SPLINE
SPL {X  -160.133, Y  +702.956, Z    +0.000, E1   -19.806, E3 +417494.548}
SPL {X  -161.979, Y  +690.023, Z    +0.000, E1   -12.991, E3 +417497.464}
SPL {X  -162.641, Y  +681.139, Z    +0.000, E1    -7.893, E3 +417499.556}
SPL {X  -162.815, Y  +674.833, Z    +0.000, E1    -4.093, E3 +417497.172}
SPL {X  -162.820, Y  +669.862, Z    +0.000, E1    -0.751, E3 +417500.390}
SPL {X  -162.820, Y  +664.572, Z    +0.000, E1    +3.252, E3 +417500.204}
SPL {X  -162.820, Y  +657.781, Z    +0.000, E1    +9.391, E3 +417498.027}
SPL {X  -162.820, Y  +648.706, Z    +0.000, E1   +17.761, E3 +417499.779}
SPL {X  -162.820, Y  +635.926, Z    +0.000, E1   +28.192, E3 +417504.606}
SPL {X  -162.820, Y  +621.673, Z    +0.000, E1   +34.265, E3 +417520.963}
SPL {X  -162.820, Y  +601.185, Z    +0.000, E1   +39.430, E3 +417547.542}
SPL {X  -162.820, Y  +599.927, Z    +0.000, E1   +35.241, E3 +417574.120}
SPL {X  -162.820, Y  +597.570, Z    +0.000, E1   +33.919, E3 +417589.849}
SPL {X  -162.820, Y  +592.692, Z    +0.000, E1   +33.779, E3 +417605.741}
SPL {X  -162.820, Y  +588.795, Z    +0.000, E1   +33.876, E3 +417617.178}
SPL {X  -162.820, Y  +584.646, Z    +0.000, E1   +33.882, E3 +417630.142}
SPL {X  -162.820, Y  +579.919, Z    +0.000, E1   +33.857, E3 +417644.930}
SPL {X  -162.820, Y  +574.615, Z    +0.000, E1   +33.920, E3 +417661.104}
SPL {X  -162.820, Y  +570.335, Z    +0.000, E1   +33.821, E3 +417674.810}
SPL {X  -162.820, Y  +565.901, Z    +0.000, E1   +33.889, E3 +417688.330}
SPL {X  -162.820, Y  +562.173, Z    +0.000, E1   +33.897, E3 +417699.621}
SPL {X  -162.820, Y  +559.395, Z    +0.000, E1   +33.796, E3 +417708.988}
SPL {X  -162.820, Y  +554.453, Z    +0.000, E1   +33.841, E3 +417724.213}
SPL {X  -162.820, Y  +549.726, Z    +0.000, E1   +33.905, E3 +417738.316}
SPL {X  -162.820, Y  +545.760, Z    +0.000, E1   +33.901, E3 +417750.712}
SPL {X  -162.820, Y  +541.668, Z    +0.000, E1   +33.787, E3 +417764.112}
SPL {X  -162.820, Y  +538.174, Z    +0.000, E1   +33.865, E3 +417774.402}
SPL {X  -162.820, Y  +534.943, Z    +0.000, E1   +33.919, E3 +417784.142}
SPL {X  -162.820, Y  +531.459, Z    +0.000, E1   +33.783, E3 +417795.799}
SPL {X  -162.820, Y  +526.783, Z    +0.000, E1   +33.870, E3 +417809.927}
SPL {X  -162.820, Y  +521.520, Z    +0.000, E1   +33.826, E3 +417826.574}
SPL {X  -162.820, Y  +516.814, Z    +0.000, E1   +33.917, E3 +417840.476}
SPL {X  -162.820, Y  +512.685, Z    +0.000, E1   +33.830, E3 +417853.918}
SPL {X  -162.820, Y  +508.888, Z    +0.000, E1   +33.871, E3 +417865.333}
SPL {X  -162.820, Y  +505.651, Z    +0.000, E1   +33.839, E3 +417875.650}
SPL {X  -162.820, Y  +500.931, Z    +0.000, E1   +34.256, E3 +417887.524}
SPL {X  -162.820, Y  +481.122, Z    +0.000, E1   +41.279, E3 +417897.788}
SPL {X  -162.820, Y  +477.698, Z    +0.000, E1   +40.353, E3 +417911.844}
SPL {X  -162.820, Y  +474.538, Z    +0.000, E1   +39.267, E3 +417926.019}
SPL {X  -162.820, Y  +472.097, Z    +0.000, E1   +38.411, E3 +417937.563}
SPL {X  -162.820, Y  +469.308, Z    +0.000, E1   +37.839, E3 +417948.367}
SPL {X  -162.820, Y  +467.216, Z    +0.000, E1   +37.215, E3 +417957.934}
SPL {X  -162.820, Y  +462.598, Z    +0.000, E1   +37.325, E3 +417969.888}
SPL {X  -162.820, Y  +457.832, Z    +0.000, E1   +37.294, E3 +417983.175}
SPL {X  -162.820, Y  +452.986, Z    +0.000, E1   +37.368, E3 +417995.908}
SPL {X  -162.820, Y  +448.311, Z    +0.000, E1   +37.333, E3 +418008.928}
SPL {X  -162.820, Y  +443.351, Z    +0.000, E1   +37.335, E3 +418022.458}
SPL {X  -162.820, Y  +438.727, Z    +0.000, E1   +37.289, E3 +418035.331}
SPL {X  -162.820, Y  +434.320, Z    +0.000, E1   +37.343, E3 +418047.040}
SPL {X  -162.820, Y  +430.091, Z    +0.000, E1   +37.424, E3 +418058.041}
SPL {X  -162.820, Y  +426.177, Z    +0.000, E1   +37.250, E3 +418069.863}
SPL {X  -162.820, Y  +421.391, Z    +0.000, E1   +37.346, E3 +418082.327}
SPL {X  -162.820, Y  +416.811, Z    +0.000, E1   +37.348, E3 +418094.861}
SPL {X  -162.820, Y  +411.860, Z    +0.000, E1   +37.402, E3 +418108.013}
SPL {X  -162.820, Y  +407.726, Z    +0.000, E1   +37.291, E3 +418119.961}
SPL {X  -162.820, Y  +403.543, Z    +0.000, E1   +37.305, E3 +418131.306}
SPL {X  -162.820, Y  +399.300, Z    +0.000, E1   +37.355, E3 +418142.590}
SPL {X  -162.820, Y  +395.182, Z    +0.000, E1   +37.347, E3 +418153.879}
SPL {X  -162.820, Y  +390.797, Z    +0.000, E1   +37.358, E3 +418165.792}
SPL {X  -162.820, Y  +385.307, Z    +0.000, E1   +37.364, E3 +418180.871}
SPL {X  -162.820, Y  +380.796, Z    +0.000, E1   +37.334, E3 +418193.158}
SPL {X  -162.785, Y  +377.133, Z    +0.000, E1   +37.299, E3 +418203.479}
SPL {X  -162.623, Y  +372.484, Z    +0.000, E1   +37.337, E3 +418215.919}
SPL {X  -162.331, Y  +367.894, Z    +0.000, E1   +37.251, E3 +418229.032}
SPL {X  -161.920, Y  +363.407, Z    +0.000, E1   +37.164, E3 +418241.766}
SPL {X  -161.341, Y  +358.603, Z    +0.000, E1   +37.117, E3 +418255.246}
SPL {X  -160.616, Y  +353.801, Z    +0.000, E1   +36.942, E3 +418269.410}
SPL {X  -159.837, Y  +349.474, Z    +0.000, E1   +36.824, E3 +418281.854}
SPL {X  -158.862, Y  +344.820, Z    +0.000, E1   +36.732, E3 +418295.217}
SPL {X  -157.959, Y  +341.011, Z    +0.000, E1   +36.448, E3 +418307.114}
SPL {X  -153.520, Y  +326.260, Z    +0.000, E1   +41.363, E3 +418315.946}
SPL {X  -150.942, Y  +319.452, Z    +0.000, E1   +36.529, E3 +418372.303}
ENDSPLINE

SPLINE
SPL {X  -159.264, Y  +346.659, Z    +0.000, E1   +22.083, E3 +418412.877}
SPL {X  -161.245, Y  +357.907, Z    +0.000, E1   +16.095, E3 +418426.310}
SPL {X  -162.697, Y  +374.161, Z    +0.000, E1    +7.119, E3 +418424.299}
SPL {X  -162.820, Y  +380.878, Z    +0.000, E1    +2.854, E3 +418427.131}
SPL {X  -162.820, Y  +385.313, Z    +0.000, E1    -0.228, E3 +418426.911}
SPL {X  -162.820, Y  +389.965, Z    +0.000, E1    -3.918, E3 +418426.279}
SPL {X  -162.820, Y  +394.532, Z    +0.000, E1    -7.849, E3 +418427.828}
SPL {X  -162.820, Y  +400.765, Z    +0.000, E1   -14.108, E3 +418425.294}
SPL {X  -162.820, Y  +411.829, Z    +0.000, E1   -24.195, E3 +418427.372}
SPL {X  -162.820, Y  +434.900, Z    +0.000, E1   -34.666, E3 +418454.736}
SPL {X  -162.820, Y  +465.440, Z    +0.000, E1   -41.264, E3 +418496.044}
ENDSPLINE

SPLINE
SPL {X  -162.820, Y  +460.175, Z    +0.000, E1   -36.098, E3 +418513.844}
ENDSPLINE

SPLINE
SPL {X  -162.820, Y  +465.690, Z    +0.000, E1   -36.140, E3 +418529.158}
SPL {X  -162.820, Y  +470.432, Z    +0.000, E1   -36.100, E3 +418543.040}
SPL {X  -162.820, Y  +475.701, Z    +0.000, E1   -36.157, E3 +418557.668}
SPL {X  -162.820, Y  +479.954, Z    +0.000, E1   -36.086, E3 +418570.208}
SPL {X  -162.820, Y  +483.976, Z    +0.000, E1   -36.049, E3 +418581.940}
SPL {X  -162.820, Y  +488.601, Z    +0.000, E1   -36.081, E3 +418595.030}
SPL {X  -162.820, Y  +493.837, Z    +0.000, E1   -36.178, E3 +418609.374}
SPL {X  -162.820, Y  +497.796, Z    +0.000, E1   -36.022, E3 +418621.558}
SPL {X  -162.820, Y  +502.146, Z    +0.000, E1   -36.123, E3 +418633.427}
SPL {X  -162.820, Y  +505.688, Z    +0.000, E1   -36.050, E3 +418643.909}
SPL {X  -162.820, Y  +509.364, Z    +0.000, E1   -36.084, E3 +418654.280}
SPL {X  -162.820, Y  +513.393, Z    +0.000, E1   -36.179, E3 +418665.136}
SPL {X  -162.820, Y  +516.436, Z    +0.000, E1   -36.094, E3 +418674.331}
SPL {X  -162.820, Y  +520.482, Z    +0.000, E1   -36.096, E3 +418685.963}
SPL {X  -162.820, Y  +524.107, Z    +0.000, E1   -36.045, E3 +418696.547}
SPL {X  -162.820, Y  +527.962, Z    +0.000, E1   -36.074, E3 +418707.480}
SPL {X  -162.820, Y  +532.253, Z    +0.000, E1   -36.170, E3 +418719.069}
SPL {X  -162.820, Y  +536.031, Z    +0.000, E1   -36.058, E3 +418730.607}
SPL {X  -162.820, Y  +541.179, Z    +0.000, E1   -36.085, E3 +418745.247}
SPL {X  -162.820, Y  +546.355, Z    +0.000, E1   -36.114, E3 +418759.792}
SPL {X  -162.820, Y  +551.776, Z    +0.000, E1   -36.108, E3 +418775.426}
SPL {X  -162.820, Y  +556.944, Z    +0.000, E1   -36.118, E3 +418789.996}
SPL {X  -162.820, Y  +561.684, Z    +0.000, E1   -36.118, E3 +418803.588}
SPL {X  -162.820, Y  +566.500, Z    +0.000, E1   -36.073, E3 +418817.591}
SPL {X  -162.820, Y  +571.734, Z    +0.000, E1   -36.094, E3 +418832.521}
SPL {X  -162.820, Y  +576.887, Z    +0.000, E1   -36.084, E3 +418847.214}
SPL {X  -162.820, Y  +581.763, Z    +0.000, E1   -36.093, E3 +418861.151}
SPL {X  -162.820, Y  +586.693, Z    +0.000, E1   -36.086, E3 +418875.256}
SPL {X  -162.820, Y  +591.665, Z    +0.000, E1   -36.045, E3 +418889.784}
SPL {X  -162.820, Y  +597.399, Z    +0.000, E1   -36.147, E3 +418905.547}
SPL {X  -162.820, Y  +602.243, Z    +0.000, E1   -36.085, E3 +418919.693}
SPL {X  -162.820, Y  +605.848, Z    +0.000, E1   -36.070, E3 +418930.014}
SPL {X  -162.820, Y  +609.375, Z    +0.000, E1   -36.084, E3 +418940.065}
SPL {X  -162.820, Y  +612.959, Z    +0.000, E1   -36.034, E3 +418950.585}
SPL {X  -162.820, Y  +616.897, Z    +0.000, E1   -36.061, E3 +418961.733}
SPL {X  -162.820, Y  +621.516, Z    +0.000, E1   -36.072, E3 +418974.932}
SPL {X  -162.820, Y  +626.243, Z    +0.000, E1   -36.105, E3 +418988.174}
SPL {X  -162.820, Y  +630.571, Z    +0.000, E1   -36.057, E3 +419000.876}
SPL {X  -162.820, Y  +635.505, Z    +0.000, E1   -36.079, E3 +419014.882}
SPL {X  -162.820, Y  +641.277, Z    +0.000, E1   -36.126, E3 +419031.175}
SPL {X  -162.820, Y  +646.320, Z    +0.000, E1   -36.078, E3 +419045.740}
SPL {X  -162.820, Y  +651.289, Z    +0.000, E1   -36.059, E3 +419060.196}
SPL {X  -162.820, Y  +656.677, Z    +0.000, E1   -36.110, E3 +419075.209}
SPL {X  -162.820, Y  +661.560, Z    +0.000, E1   -36.068, E3 +419089.472}
SPL {X  -162.820, Y  +666.386, Z    +0.000, E1   -36.048, E3 +419103.357}
SPL {X  -162.820, Y  +672.345, Z    +0.000, E1   -36.097, E3 +419120.297}
SPL {X  -162.761, Y  +677.889, Z    +0.000, E1   -36.122, E3 +419135.762}
SPL {X  -162.577, Y  +682.401, Z    +0.000, E1   -36.021, E3 +419149.379}
SPL {X  -162.187, Y  +687.846, Z    +0.000, E1   -36.007, E3 +419165.048}
SPL {X  -161.667, Y  +692.839, Z    +0.000, E1   -35.918, E3 +419179.813}
SPL {X  -161.078, Y  +697.256, Z    +0.000, E1   -35.797, E3 +419193.149}
SPL {X  -160.313, Y  +701.964, Z    +0.000, E1   -35.709, E3 +419207.224}
SPL {X  -159.317, Y  +707.091, Z    +0.000, E1   -35.482, E3 +419223.248}
SPL {X  -158.510, Y  +710.714, Z    +0.000, E1   -35.230, E3 +419234.959}
SPL {X  -155.691, Y  +721.150, Z    +0.000, E1   -39.118, E3 +419240.344}
SPL {X  -154.394, Y  +725.200, Z    +0.000, E1   -39.595, E3 +419247.610}
SPL {X  -152.141, Y  +731.494, Z    +0.000, E1   -35.181, E3 +419302.861}
ENDSPLINE

SPLINE
SPL {X  -160.133, Y  +702.956, Z    +0.000, E1   -19.806, E3 +419346.399}
SPL {X  -161.979, Y  +690.023, Z    +0.000, E1   -12.991, E3 +419349.316}
SPL {X  -162.641, Y  +681.139, Z    +0.000, E1    -7.893, E3 +419351.408}
SPL {X  -162.820, Y  +673.062, Z    +0.000, E1    -2.992, E3 +419350.375}
SPL {X  -162.820, Y  +666.731, Z    +0.000, E1    +1.545, E3 +419352.005}
SPL {X  -162.820, Y  +660.758, Z    +0.000, E1    +6.523, E3 +419351.715}
SPL {X  -162.820, Y  +650.583, Z    +0.000, E1   +16.035, E3 +419350.688}
SPL {X  -162.820, Y  +629.267, Z    +0.000, E1   +31.872, E3 +419361.836}
SPL {X  -162.820, Y  +620.680, Z    +0.000, E1   +34.107, E3 +419375.886}
SPL {X  -162.820, Y  +609.002, Z    +0.000, E1   +38.458, E3 +419386.037}
SPL {X  -162.820, Y  +596.392, Z    +0.000, E1   +37.895, E3 +419419.506}
ENDSPLINE

SPLINE
SPL {X  -162.820, Y  +599.924, Z    +0.000, E1   +33.992, E3 +419433.880}
ENDSPLINE

SPLINE
SPL {X  -162.820, Y  +595.170, Z    +0.000, E1   +33.784, E3 +419449.928}
SPL {X  -162.820, Y  +589.785, Z    +0.000, E1   +33.904, E3 +419465.925}
SPL {X  -162.820, Y  +584.646, Z    +0.000, E1   +33.882, E3 +419481.994}
SPL {X  -162.820, Y  +579.919, Z    +0.000, E1   +33.857, E3 +419496.782}
SPL {X  -162.820, Y  +574.615, Z    +0.000, E1   +33.920, E3 +419512.956}
SPL {X  -162.820, Y  +570.335, Z    +0.000, E1   +33.821, E3 +419526.662}
SPL {X  -162.820, Y  +565.901, Z    +0.000, E1   +33.889, E3 +419540.182}
SPL {X  -162.820, Y  +560.226, Z    +0.000, E1   +33.868, E3 +419557.967}
SPL {X  -162.820, Y  +554.453, Z    +0.000, E1   +33.841, E3 +419576.065}
SPL {X  -162.820, Y  +549.726, Z    +0.000, E1   +33.905, E3 +419590.168}
SPL {X  -162.820, Y  +545.760, Z    +0.000, E1   +33.901, E3 +419602.564}
SPL {X  -162.820, Y  +541.668, Z    +0.000, E1   +33.787, E3 +419615.964}
SPL {X  -162.820, Y  +538.174, Z    +0.000, E1   +33.865, E3 +419626.254}
SPL {X  -162.820, Y  +534.943, Z    +0.000, E1   +33.919, E3 +419635.994}
SPL {X  -162.820, Y  +530.273, Z    +0.000, E1   +33.855, E3 +419651.023}
SPL {X  -162.820, Y  +524.900, Z    +0.000, E1   +33.820, E3 +419667.924}
SPL {X  -162.820, Y  +520.532, Z    +0.000, E1   +33.805, E3 +419681.491}
SPL {X  -162.820, Y  +516.814, Z    +0.000, E1   +33.917, E3 +419692.327}
SPL {X  -162.820, Y  +512.685, Z    +0.000, E1   +33.830, E3 +419705.770}
SPL {X  -162.820, Y  +508.888, Z    +0.000, E1   +33.871, E3 +419717.185}
SPL {X  -162.820, Y  +505.651, Z    +0.000, E1   +33.839, E3 +419727.502}
SPL {X  -162.820, Y  +500.931, Z    +0.000, E1   +34.256, E3 +419739.375}
SPL {X  -162.820, Y  +481.122, Z    +0.000, E1   +41.279, E3 +419749.640}
SPL {X  -162.820, Y  +478.698, Z    +0.000, E1   +40.526, E3 +419759.989}
SPL {X  -162.820, Y  +475.203, Z    +0.000, E1   +39.596, E3 +419774.448}
SPL {X  -162.820, Y  +472.097, Z    +0.000, E1   +38.411, E3 +419789.415}
SPL {X  -162.820, Y  +469.308, Z    +0.000, E1   +37.839, E3 +419800.219}
SPL {X  -162.820, Y  +467.216, Z    +0.000, E1   +37.215, E3 +419809.786}
SPL {X  -162.820, Y  +462.598, Z    +0.000, E1   +37.325, E3 +419821.740}
SPL {X  -162.820, Y  +457.832, Z    +0.000, E1   +37.294, E3 +419835.027}
SPL {X  -162.820, Y  +452.986, Z    +0.000, E1   +37.368, E3 +419847.760}
SPL {X  -162.820, Y  +448.311, Z    +0.000, E1   +37.333, E3 +419860.780}
SPL {X  -162.820, Y  +443.351, Z    +0.000, E1   +37.335, E3 +419874.310}
SPL {X  -162.820, Y  +438.727, Z    +0.000, E1   +37.289, E3 +419887.182}
SPL {X  -162.820, Y  +434.320, Z    +0.000, E1   +37.343, E3 +419898.892}
SPL {X  -162.820, Y  +430.091, Z    +0.000, E1   +37.424, E3 +419909.892}
SPL {X  -162.820, Y  +426.177, Z    +0.000, E1   +37.250, E3 +419921.715}
SPL {X  -162.820, Y  +420.241, Z    +0.000, E1   +37.355, E3 +419937.422}
SPL {X  -162.820, Y  +415.595, Z    +0.000, E1   +37.375, E3 +419949.762}
SPL {X  -162.820, Y  +411.860, Z    +0.000, E1   +37.402, E3 +419959.865}
SPL {X  -162.820, Y  +407.726, Z    +0.000, E1   +37.291, E3 +419971.812}
SPL {X  -162.820, Y  +403.543, Z    +0.000, E1   +37.305, E3 +419983.158}
SPL {X  -162.820, Y  +399.300, Z    +0.000, E1   +37.355, E3 +419994.442}
SPL {X  -162.820, Y  +395.182, Z    +0.000, E1   +37.347, E3 +420005.731}
SPL {X  -162.820, Y  +390.797, Z    +0.000, E1   +37.358, E3 +420017.643}
SPL {X  -162.820, Y  +386.671, Z    +0.000, E1   +37.363, E3 +420028.824}
SPL {X  -162.820, Y  +382.174, Z    +0.000, E1   +37.329, E3 +420041.402}
SPL {X  -162.785, Y  +377.133, Z    +0.000, E1   +37.299, E3 +420055.331}
SPL {X  -162.623, Y  +372.484, Z    +0.000, E1   +37.337, E3 +420067.771}
SPL {X  -162.331, Y  +367.894, Z    +0.000, E1   +37.251, E3 +420080.883}
SPL {X  -161.920, Y  +363.407, Z    +0.000, E1   +37.164, E3 +420093.617}
SPL {X  -161.482, Y  +359.669, Z    +0.000, E1   +37.064, E3 +420104.402}
SPL {X  -160.943, Y  +355.851, Z    +0.000, E1   +37.136, E3 +420114.389}
SPL {X  -160.493, Y  +353.069, Z    +0.000, E1   +36.789, E3 +420124.041}
SPL {X  -159.837, Y  +349.474, Z    +0.000, E1   +36.824, E3 +420133.706}
SPL {X  -159.171, Y  +346.224, Z    +0.000, E1   +36.747, E3 +420142.983}
SPL {X  -158.248, Y  +342.188, Z    +0.000, E1   +36.583, E3 +420155.145}
SPL {X  -153.520, Y  +326.260, Z    +0.000, E1   +41.363, E3 +420167.798}
SPL {X  -150.942, Y  +319.452, Z    +0.000, E1   +36.529, E3 +420224.155}
ENDSPLINE

SPLINE
SPL {X  -159.264, Y  +346.659, Z    +0.000, E1   +22.083, E3 +420264.729}
SPL {X  -161.245, Y  +357.907, Z    +0.000, E1   +16.095, E3 +420278.162}
SPL {X  -162.746, Y  +375.590, Z    +0.000, E1    +6.280, E3 +420277.750}
SPL {X  -162.820, Y  +384.478, Z    +0.000, E1    +0.434, E3 +420278.419}
SPL {X  -162.820, Y  +389.965, Z    +0.000, E1    -3.918, E3 +420278.131}
SPL {X  -162.820, Y  +394.532, Z    +0.000, E1    -7.849, E3 +420279.679}
SPL {X  -162.820, Y  +400.765, Z    +0.000, E1   -14.108, E3 +420277.146}
SPL {X  -162.820, Y  +411.829, Z    +0.000, E1   -24.195, E3 +420279.224}
SPL {X  -162.820, Y  +434.900, Z    +0.000, E1   -34.666, E3 +420306.588}
SPL {X  -162.820, Y  +465.031, Z    +0.000, E1   -41.710, E3 +420344.261}
SPL {X  -162.820, Y  +465.893, Z    +0.000, E1   -40.572, E3 +420352.790}
ENDSPLINE

SPLINE
SPL {X  -162.820, Y  +458.794, Z    +0.000, E1   -36.100, E3 +420361.519}
ENDSPLINE

SPLINE
SPL {X  -162.820, Y  +461.779, Z    +0.000, E1   -35.988, E3 +420370.715}
SPL {X  -162.820, Y  +465.690, Z    +0.000, E1   -36.140, E3 +420381.010}
SPL {X  -162.820, Y  +470.432, Z    +0.000, E1   -36.100, E3 +420394.892}
SPL {X  -162.820, Y  +475.701, Z    +0.000, E1   -36.157, E3 +420409.520}
SPL {X  -162.820, Y  +479.954, Z    +0.000, E1   -36.086, E3 +420422.060}
SPL {X  -162.820, Y  +483.976, Z    +0.000, E1   -36.049, E3 +420433.792}
SPL {X  -162.820, Y  +488.601, Z    +0.000, E1   -36.081, E3 +420446.882}
SPL {X  -162.820, Y  +493.837, Z    +0.000, E1   -36.178, E3 +420461.225}
SPL {X  -162.820, Y  +498.932, Z    +0.000, E1   -36.079, E3 +420476.430}
SPL {X  -162.820, Y  +504.528, Z    +0.000, E1   -36.109, E3 +420492.226}
SPL {X  -162.820, Y  +509.364, Z    +0.000, E1   -36.084, E3 +420506.132}
SPL {X  -162.820, Y  +515.001, Z    +0.000, E1   -36.183, E3 +420521.769}
SPL {X  -162.820, Y  +520.482, Z    +0.000, E1   -36.096, E3 +420537.815}
SPL {X  -162.820, Y  +525.226, Z    +0.000, E1   -36.081, E3 +420551.483}
SPL {X  -162.820, Y  +530.908, Z    +0.000, E1   -36.155, E3 +420567.340}
SPL {X  -162.820, Y  +536.031, Z    +0.000, E1   -36.058, E3 +420582.459}
SPL {X  -162.820, Y  +541.179, Z    +0.000, E1   -36.085, E3 +420597.099}
SPL {X  -162.820, Y  +546.355, Z    +0.000, E1   -36.114, E3 +420611.644}
SPL {X  -162.820, Y  +551.776, Z    +0.000, E1   -36.108, E3 +420627.278}
SPL {X  -162.820, Y  +556.944, Z    +0.000, E1   -36.118, E3 +420641.848}
SPL {X  -162.820, Y  +561.684, Z    +0.000, E1   -36.118, E3 +420655.440}
SPL {X  -162.820, Y  +566.500, Z    +0.000, E1   -36.073, E3 +420669.443}
SPL {X  -162.820, Y  +571.734, Z    +0.000, E1   -36.094, E3 +420684.373}
SPL {X  -162.820, Y  +576.887, Z    +0.000, E1   -36.084, E3 +420699.066}
SPL {X  -162.820, Y  +581.763, Z    +0.000, E1   -36.093, E3 +420713.003}
SPL {X  -162.820, Y  +586.693, Z    +0.000, E1   -36.086, E3 +420727.108}
SPL {X  -162.820, Y  +590.250, Z    +0.000, E1   -36.075, E3 +420737.226}
SPL {X  -162.820, Y  +594.470, Z    +0.000, E1   -36.080, E3 +420749.457}
SPL {X  -162.820, Y  +598.788, Z    +0.000, E1   -36.102, E3 +420761.478}
SPL {X  -162.820, Y  +602.243, Z    +0.000, E1   -36.085, E3 +420771.545}
SPL {X  -162.820, Y  +605.848, Z    +0.000, E1   -36.070, E3 +420781.866}
SPL {X  -162.820, Y  +609.375, Z    +0.000, E1   -36.084, E3 +420791.917}
SPL {X  -162.820, Y  +612.959, Z    +0.000, E1   -36.034, E3 +420802.437}
SPL {X  -162.820, Y  +616.897, Z    +0.000, E1   -36.061, E3 +420813.584}
SPL {X  -162.820, Y  +621.516, Z    +0.000, E1   -36.072, E3 +420826.783}
SPL {X  -162.820, Y  +626.243, Z    +0.000, E1   -36.105, E3 +420840.026}
SPL {X  -162.820, Y  +630.571, Z    +0.000, E1   -36.057, E3 +420852.728}
SPL {X  -162.820, Y  +635.505, Z    +0.000, E1   -36.079, E3 +420866.734}
SPL {X  -162.820, Y  +641.277, Z    +0.000, E1   -36.126, E3 +420883.027}
SPL {X  -162.820, Y  +646.320, Z    +0.000, E1   -36.078, E3 +420897.592}
SPL {X  -162.820, Y  +651.289, Z    +0.000, E1   -36.059, E3 +420912.048}
SPL {X  -162.820, Y  +656.677, Z    +0.000, E1   -36.110, E3 +420927.061}
SPL {X  -162.820, Y  +661.560, Z    +0.000, E1   -36.068, E3 +420941.324}
SPL {X  -162.820, Y  +666.386, Z    +0.000, E1   -36.048, E3 +420955.209}
SPL {X  -162.820, Y  +672.345, Z    +0.000, E1   -36.097, E3 +420972.149}
SPL {X  -162.761, Y  +677.889, Z    +0.000, E1   -36.122, E3 +420987.614}
SPL {X  -162.577, Y  +682.401, Z    +0.000, E1   -36.021, E3 +421001.230}
SPL {X  -162.187, Y  +687.846, Z    +0.000, E1   -36.007, E3 +421016.899}
SPL {X  -161.667, Y  +692.839, Z    +0.000, E1   -35.918, E3 +421031.665}
SPL {X  -160.925, Y  +698.267, Z    +0.000, E1   -35.816, E3 +421047.927}
SPL {X  -160.151, Y  +702.861, Z    +0.000, E1   -35.643, E3 +421061.897}
SPL {X  -159.317, Y  +707.091, Z    +0.000, E1   -35.482, E3 +421075.100}
SPL {X  -158.510, Y  +710.714, Z    +0.000, E1   -35.230, E3 +421086.811}
SPL {X  -155.037, Y  +723.239, Z    +0.000, E1   -39.382, E3 +421095.907}
SPL {X  -152.141, Y  +731.494, Z    +0.000, E1   -35.181, E3 +421154.713}
ENDSPLINE

SPLINE
SPL {X  -160.133, Y  +702.956, Z    +0.000, E1   -19.806, E3 +421198.251}
SPL {X  -161.979, Y  +690.023, Z    +0.000, E1   -12.991, E3 +421201.168}
SPL {X  -162.641, Y  +681.139, Z    +0.000, E1    -7.893, E3 +421203.260}
SPL {X  -162.820, Y  +673.062, Z    +0.000, E1    -2.992, E3 +421202.227}
SPL {X  -162.820, Y  +665.516, Z    +0.000, E1    +2.410, E3 +421204.067}
SPL {X  -162.820, Y  +657.781, Z    +0.000, E1    +9.391, E3 +421201.731}
SPL {X  -162.820, Y  +648.706, Z    +0.000, E1   +17.761, E3 +421203.482}
SPL {X  -162.820, Y  +629.267, Z    +0.000, E1   +31.872, E3 +421213.688}
SPL {X  -162.820, Y  +617.390, Z    +0.000, E1   +35.413, E3 +421230.618}
SPL {X  -162.820, Y  +596.392, Z    +0.000, E1   +37.895, E3 +421271.358}
ENDSPLINE

SPLINE
SPL {X  -162.820, Y  +601.432, Z    +0.000, E1   +34.026, E3 +421280.656}
ENDSPLINE

SPLINE
SPL {X  -162.820, Y  +597.570, Z    +0.000, E1   +33.919, E3 +421293.553}
SPL {X  -162.820, Y  +592.692, Z    +0.000, E1   +33.779, E3 +421309.445}
SPL {X  -162.820, Y  +588.795, Z    +0.000, E1   +33.876, E3 +421320.882}
SPL {X  -162.820, Y  +585.519, Z    +0.000, E1   +33.888, E3 +421330.966}
SPL {X  -162.820, Y  +582.066, Z    +0.000, E1   +33.857, E3 +421341.901}
SPL {X  -162.820, Y  +577.919, Z    +0.000, E1   +33.841, E3 +421354.954}
SPL {X  -162.820, Y  +573.566, Z    +0.000, E1   +33.899, E3 +421368.029}
SPL {X  -162.820, Y  +569.298, Z    +0.000, E1   +33.851, E3 +421381.670}
SPL {X  -162.820, Y  +563.983, Z    +0.000, E1   +33.916, E3 +421397.811}
SPL {X  -162.820, Y  +559.395, Z    +0.000, E1   +33.796, E3 +421412.692}
SPL {X  -162.820, Y  +554.453, Z    +0.000, E1   +33.841, E3 +421427.917}
SPL {X  -162.820, Y  +549.726, Z    +0.000, E1   +33.905, E3 +421442.020}
SPL {X  -162.820, Y  +545.760, Z    +0.000, E1   +33.901, E3 +421454.416}
SPL {X  -162.820, Y  +541.668, Z    +0.000, E1   +33.787, E3 +421467.816}
SPL {X  -162.820, Y  +538.174, Z    +0.000, E1   +33.865, E3 +421478.106}
SPL {X  -162.820, Y  +534.943, Z    +0.000, E1   +33.919, E3 +421487.846}
SPL {X  -162.820, Y  +530.273, Z    +0.000, E1   +33.855, E3 +421502.875}
SPL {X  -162.820, Y  +524.900, Z    +0.000, E1   +33.820, E3 +421519.776}
SPL {X  -162.820, Y  +520.532, Z    +0.000, E1   +33.805, E3 +421533.343}
SPL {X  -162.820, Y  +516.814, Z    +0.000, E1   +33.917, E3 +421544.179}
SPL {X  -162.820, Y  +512.685, Z    +0.000, E1   +33.830, E3 +421557.622}
SPL {X  -162.820, Y  +508.888, Z    +0.000, E1   +33.871, E3 +421569.037}
SPL {X  -162.820, Y  +505.651, Z    +0.000, E1   +33.839, E3 +421579.354}
SPL {X  -162.820, Y  +500.931, Z    +0.000, E1   +34.256, E3 +421591.227}
SPL {X  -162.820, Y  +481.122, Z    +0.000, E1   +41.279, E3 +421601.492}
SPL {X  -162.820, Y  +477.698, Z    +0.000, E1   +40.353, E3 +421615.548}
SPL {X  -162.820, Y  +474.538, Z    +0.000, E1   +39.267, E3 +421629.723}
SPL {X  -162.820, Y  +472.097, Z    +0.000, E1   +38.411, E3 +421641.267}
SPL {X  -162.820, Y  +469.308, Z    +0.000, E1   +37.839, E3 +421652.071}
SPL {X  -162.820, Y  +467.216, Z    +0.000, E1   +37.215, E3 +421661.638}
SPL {X  -162.820, Y  +462.598, Z    +0.000, E1   +37.325, E3 +421673.592}
SPL {X  -162.820, Y  +457.832, Z    +0.000, E1   +37.294, E3 +421686.878}
SPL {X  -162.820, Y  +452.986, Z    +0.000, E1   +37.368, E3 +421699.612}
SPL {X  -162.820, Y  +448.311, Z    +0.000, E1   +37.333, E3 +421712.632}
SPL {X  -162.820, Y  +443.351, Z    +0.000, E1   +37.335, E3 +421726.162}
SPL {X  -162.820, Y  +438.727, Z    +0.000, E1   +37.289, E3 +421739.034}
SPL {X  -162.820, Y  +434.320, Z    +0.000, E1   +37.343, E3 +421750.744}
SPL {X  -162.820, Y  +430.091, Z    +0.000, E1   +37.424, E3 +421761.744}
SPL {X  -162.820, Y  +426.177, Z    +0.000, E1   +37.250, E3 +421773.567}
SPL {X  -162.820, Y  +421.391, Z    +0.000, E1   +37.346, E3 +421786.031}
SPL {X  -162.820, Y  +416.811, Z    +0.000, E1   +37.348, E3 +421798.565}
SPL {X  -162.820, Y  +411.860, Z    +0.000, E1   +37.402, E3 +421811.717}
SPL {X  -162.820, Y  +407.726, Z    +0.000, E1   +37.291, E3 +421823.664}
SPL {X  -162.820, Y  +403.543, Z    +0.000, E1   +37.305, E3 +421835.010}
SPL {X  -162.820, Y  +399.300, Z    +0.000, E1   +37.355, E3 +421846.294}
SPL {X  -162.820, Y  +395.182, Z    +0.000, E1   +37.347, E3 +421857.583}
SPL {X  -162.820, Y  +390.797, Z    +0.000, E1   +37.358, E3 +421869.495}
SPL {X  -162.820, Y  +386.671, Z    +0.000, E1   +37.363, E3 +421880.676}
SPL {X  -162.820, Y  +382.174, Z    +0.000, E1   +37.329, E3 +421893.254}
SPL {X  -162.785, Y  +377.133, Z    +0.000, E1   +37.299, E3 +421907.183}
SPL {X  -162.576, Y  +371.586, Z    +0.000, E1   +37.322, E3 +421922.296}
SPL {X  -162.256, Y  +366.963, Z    +0.000, E1   +37.251, E3 +421935.184}
SPL {X  -161.920, Y  +363.407, Z    +0.000, E1   +37.164, E3 +421945.469}
SPL {X  -161.341, Y  +358.603, Z    +0.000, E1   +37.117, E3 +421958.950}
SPL {X  -160.616, Y  +353.801, Z    +0.000, E1   +36.942, E3 +421973.114}
SPL {X  -159.837, Y  +349.474, Z    +0.000, E1   +36.824, E3 +421985.558}
SPL {X  -158.862, Y  +344.820, Z    +0.000, E1   +36.732, E3 +421998.921}
SPL {X  -157.959, Y  +341.011, Z    +0.000, E1   +36.448, E3 +422010.818}
SPL {X  -153.520, Y  +326.260, Z    +0.000, E1   +41.363, E3 +422019.650}
SPL {X  -150.942, Y  +319.452, Z    +0.000, E1   +36.529, E3 +422076.007}
ENDSPLINE

SPLINE
SPL {X  -159.264, Y  +346.659, Z    +0.000, E1   +22.083, E3 +422116.581}
SPL {X  -161.245, Y  +357.907, Z    +0.000, E1   +16.095, E3 +422130.014}
SPL {X  -162.697, Y  +374.161, Z    +0.000, E1    +7.119, E3 +422128.003}
SPL {X  -162.820, Y  +380.878, Z    +0.000, E1    +2.854, E3 +422130.834}
SPL {X  -162.820, Y  +385.313, Z    +0.000, E1    -0.228, E3 +422130.615}
SPL {X  -162.820, Y  +389.965, Z    +0.000, E1    -3.918, E3 +422129.983}
SPL {X  -162.820, Y  +394.532, Z    +0.000, E1    -7.849, E3 +422131.531}
SPL {X  -162.820, Y  +400.765, Z    +0.000, E1   -14.108, E3 +422128.998}
SPL {X  -162.820, Y  +411.829, Z    +0.000, E1   -24.195, E3 +422131.076}
SPL {X  -162.820, Y  +434.900, Z    +0.000, E1   -34.666, E3 +422158.440}
SPL {X  -162.820, Y  +465.440, Z    +0.000, E1   -41.264, E3 +422199.748}
ENDSPLINE

SPLINE
SPL {X  -162.820, Y  +460.175, Z    +0.000, E1   -36.098, E3 +422217.547}
ENDSPLINE

SPLINE
SPL {X  -162.820, Y  +467.031, Z    +0.000, E1   -36.178, E3 +422236.637}
SPL {X  -162.820, Y  +471.524, Z    +0.000, E1   -36.022, E3 +422250.190}
SPL {X  -162.820, Y  +475.701, Z    +0.000, E1   -36.157, E3 +422261.371}
SPL {X  -162.820, Y  +479.954, Z    +0.000, E1   -36.086, E3 +422273.912}
SPL {X  -162.820, Y  +483.976, Z    +0.000, E1   -36.049, E3 +422285.644}
SPL {X  -162.820, Y  +488.601, Z    +0.000, E1   -36.081, E3 +422298.734}
SPL {X  -162.820, Y  +493.837, Z    +0.000, E1   -36.178, E3 +422313.077}
SPL {X  -162.820, Y  +497.796, Z    +0.000, E1   -36.022, E3 +422325.262}
SPL {X  -162.820, Y  +502.146, Z    +0.000, E1   -36.123, E3 +422337.131}
SPL {X  -162.820, Y  +505.688, Z    +0.000, E1   -36.050, E3 +422347.613}
SPL {X  -162.820, Y  +509.364, Z    +0.000, E1   -36.084, E3 +422357.983}
SPL {X  -162.820, Y  +515.001, Z    +0.000, E1   -36.183, E3 +422373.621}
SPL {X  -162.820, Y  +520.482, Z    +0.000, E1   -36.096, E3 +422389.667}
SPL {X  -162.820, Y  +524.107, Z    +0.000, E1   -36.045, E3 +422400.251}
SPL {X  -162.820, Y  +527.962, Z    +0.000, E1   -36.074, E3 +422411.183}
SPL {X  -162.820, Y  +532.253, Z    +0.000, E1   -36.170, E3 +422422.772}
SPL {X  -162.820, Y  +536.031, Z    +0.000, E1   -36.058, E3 +422434.311}
SPL {X  -162.820, Y  +540.096, Z    +0.000, E1   -36.040, E3 +422446.009}
SPL {X  -162.820, Y  +545.472, Z    +0.000, E1   -36.142, E3 +422460.946}
SPL {X  -162.820, Y  +551.776, Z    +0.000, E1   -36.108, E3 +422479.129}
SPL {X  -162.820, Y  +558.272, Z    +0.000, E1   -36.170, E3 +422497.338}
SPL {X  -162.820, Y  +562.721, Z    +0.000, E1   -36.046, E3 +422510.563}
SPL {X  -162.820, Y  +566.500, Z    +0.000, E1   -36.073, E3 +422521.295}
SPL {X  -162.820, Y  +571.734, Z    +0.000, E1   -36.094, E3 +422536.224}
SPL {X  -162.820, Y  +576.887, Z    +0.000, E1   -36.084, E3 +422550.918}
SPL {X  -162.820, Y  +581.763, Z    +0.000, E1   -36.093, E3 +422564.855}
SPL {X  -162.820, Y  +586.693, Z    +0.000, E1   -36.086, E3 +422578.960}
SPL {X  -162.820, Y  +590.250, Z    +0.000, E1   -36.075, E3 +422589.078}
SPL {X  -162.820, Y  +594.470, Z    +0.000, E1   -36.080, E3 +422601.309}
SPL {X  -162.820, Y  +598.788, Z    +0.000, E1   -36.102, E3 +422613.330}
SPL {X  -162.820, Y  +602.243, Z    +0.000, E1   -36.085, E3 +422623.397}
SPL {X  -162.820, Y  +606.975, Z    +0.000, E1   -36.102, E3 +422636.842}
SPL {X  -162.820, Y  +611.980, Z    +0.000, E1   -36.072, E3 +422651.388}
SPL {X  -162.820, Y  +616.897, Z    +0.000, E1   -36.061, E3 +422665.436}
SPL {X  -162.820, Y  +620.590, Z    +0.000, E1   -36.079, E3 +422675.831}
SPL {X  -162.820, Y  +625.276, Z    +0.000, E1   -36.104, E3 +422689.248}
SPL {X  -162.820, Y  +630.571, Z    +0.000, E1   -36.057, E3 +422704.580}
SPL {X  -162.820, Y  +634.189, Z    +0.000, E1   -36.065, E3 +422714.774}
SPL {X  -162.820, Y  +638.473, Z    +0.000, E1   -36.098, E3 +422727.010}
SPL {X  -162.820, Y  +642.832, Z    +0.000, E1   -36.091, E3 +422739.336}
SPL {X  -162.820, Y  +646.320, Z    +0.000, E1   -36.078, E3 +422749.444}
SPL {X  -162.820, Y  +651.289, Z    +0.000, E1   -36.059, E3 +422763.900}
SPL {X  -162.820, Y  +656.677, Z    +0.000, E1   -36.110, E3 +422778.913}
SPL {X  -162.820, Y  +661.560, Z    +0.000, E1   -36.068, E3 +422793.176}
SPL {X  -162.820, Y  +666.386, Z    +0.000, E1   -36.048, E3 +422807.060}
SPL {X  -162.820, Y  +672.345, Z    +0.000, E1   -36.097, E3 +422824.001}
SPL {X  -162.761, Y  +677.889, Z    +0.000, E1   -36.122, E3 +422839.466}
SPL {X  -162.577, Y  +682.401, Z    +0.000, E1   -36.021, E3 +422853.082}
SPL {X  -162.296, Y  +686.558, Z    +0.000, E1   -35.952, E3 +422865.273}
SPL {X  -161.948, Y  +690.331, Z    +0.000, E1   -35.960, E3 +422876.071}
SPL {X  -161.544, Y  +693.846, Z    +0.000, E1   -35.908, E3 +422886.346}
SPL {X  -160.925, Y  +698.267, Z    +0.000, E1   -35.816, E3 +422899.778}
SPL {X  -160.151, Y  +702.861, Z    +0.000, E1   -35.643, E3 +422913.748}
SPL {X  -159.317, Y  +707.091, Z    +0.000, E1   -35.482, E3 +422926.952}
SPL {X  -158.510, Y  +710.714, Z    +0.000, E1   -35.230, E3 +422938.663}
SPL {X  -155.037, Y  +723.239, Z    +0.000, E1   -39.382, E3 +422947.759}
SPL {X  -152.141, Y  +731.494, Z    +0.000, E1   -35.181, E3 +423006.565}
ENDSPLINE

SPLINE
SPL {X  -160.133, Y  +702.956, Z    +0.000, E1   -19.806, E3 +423050.103}
SPL {X  -161.979, Y  +690.023, Z    +0.000, E1   -12.991, E3 +423053.020}
SPL {X  -162.641, Y  +681.139, Z    +0.000, E1    -7.893, E3 +423055.112}
SPL {X  -162.820, Y  +673.062, Z    +0.000, E1    -2.992, E3 +423054.079}
SPL {X  -162.820, Y  +666.731, Z    +0.000, E1    +1.545, E3 +423055.709}
SPL {X  -162.820, Y  +660.758, Z    +0.000, E1    +6.523, E3 +423055.419}
SPL {X  -162.820, Y  +650.583, Z    +0.000, E1   +16.035, E3 +423054.392}
SPL {X  -162.820, Y  +629.267, Z    +0.000, E1   +31.872, E3 +423065.540}
SPL {X  -162.820, Y  +617.390, Z    +0.000, E1   +35.413, E3 +423082.469}
SPL {X  -162.820, Y  +596.392, Z    +0.000, E1   +37.895, E3 +423123.210}
ENDSPLINE

SPLINE
SPL {X  -162.820, Y  +599.924, Z    +0.000, E1   +33.992, E3 +423137.583}
ENDSPLINE

SPLINE
SPL {X  -162.820, Y  +595.170, Z    +0.000, E1   +33.784, E3 +423153.632}
SPL {X  -162.820, Y  +589.785, Z    +0.000, E1   +33.904, E3 +423169.629}
SPL {X  -162.820, Y  +585.519, Z    +0.000, E1   +33.888, E3 +423182.818}
SPL {X  -162.820, Y  +582.066, Z    +0.000, E1   +33.857, E3 +423193.752}
SPL {X  -162.820, Y  +577.919, Z    +0.000, E1   +33.841, E3 +423206.806}
SPL {X  -162.820, Y  +573.566, Z    +0.000, E1   +33.899, E3 +423219.881}
SPL {X  -162.820, Y  +569.298, Z    +0.000, E1   +33.851, E3 +423233.522}
SPL {X  -162.820, Y  +565.024, Z    +0.000, E1   +33.872, E3 +423246.578}
SPL {X  -162.820, Y  +560.226, Z    +0.000, E1   +33.868, E3 +423261.671}
SPL {X  -162.820, Y  +556.206, Z    +0.000, E1   +33.843, E3 +423274.071}
SPL {X  -162.820, Y  +553.486, Z    +0.000, E1   +33.777, E3 +423283.017}
SPL {X  -162.820, Y  +549.726, Z    +0.000, E1   +33.905, E3 +423293.872}
SPL {X  -162.820, Y  +545.760, Z    +0.000, E1   +33.901, E3 +423306.268}
SPL {X  -162.820, Y  +541.668, Z    +0.000, E1   +33.787, E3 +423319.668}
SPL {X  -162.820, Y  +538.174, Z    +0.000, E1   +33.865, E3 +423329.957}
SPL {X  -162.820, Y  +534.943, Z    +0.000, E1   +33.919, E3 +423339.698}
SPL {X  -162.820, Y  +531.459, Z    +0.000, E1   +33.783, E3 +423351.355}
SPL {X  -162.820, Y  +526.783, Z    +0.000, E1   +33.870, E3 +423365.483}
SPL {X  -162.820, Y  +521.520, Z    +0.000, E1   +33.826, E3 +423382.130}
SPL {X  -162.820, Y  +516.814, Z    +0.000, E1   +33.917, E3 +423396.031}
SPL {X  -162.820, Y  +512.685, Z    +0.000, E1   +33.830, E3 +423409.474}
SPL {X  -162.820, Y  +508.888, Z    +0.000, E1   +33.871, E3 +423420.889}
SPL {X  -162.820, Y  +505.651, Z    +0.000, E1   +33.839, E3 +423431.206}
SPL {X  -162.820, Y  +500.931, Z    +0.000, E1   +34.256, E3 +423443.079}
SPL {X  -162.820, Y  +481.122, Z    +0.000, E1   +41.279, E3 +423453.344}
SPL {X  -162.820, Y  +478.698, Z    +0.000, E1   +40.526, E3 +423463.693}
SPL {X  -162.820, Y  +476.364, Z    +0.000, E1   +39.976, E3 +423472.654}
SPL {X  -162.820, Y  +473.851, Z    +0.000, E1   +39.059, E3 +423484.791}
SPL {X  -162.820, Y  +470.157, Z    +0.000, E1   +38.016, E3 +423500.728}
SPL {X  -162.820, Y  +467.216, Z    +0.000, E1   +37.215, E3 +423513.489}
SPL {X  -162.820, Y  +462.598, Z    +0.000, E1   +37.325, E3 +423525.444}
SPL {X  -162.820, Y  +457.832, Z    +0.000, E1   +37.294, E3 +423538.730}
SPL {X  -162.820, Y  +452.986, Z    +0.000, E1   +37.368, E3 +423551.464}
SPL {X  -162.820, Y  +448.311, Z    +0.000, E1   +37.333, E3 +423564.484}
SPL {X  -162.820, Y  +443.351, Z    +0.000, E1   +37.335, E3 +423578.014}
SPL {X  -162.820, Y  +438.727, Z    +0.000, E1   +37.289, E3 +423590.886}
SPL {X  -162.820, Y  +434.320, Z    +0.000, E1   +37.343, E3 +423602.596}
SPL {X  -162.820, Y  +430.091, Z    +0.000, E1   +37.424, E3 +423613.596}
SPL {X  -162.820, Y  +426.177, Z    +0.000, E1   +37.250, E3 +423625.419}
SPL {X  -162.820, Y  +421.391, Z    +0.000, E1   +37.346, E3 +423637.883}
SPL {X  -162.820, Y  +416.811, Z    +0.000, E1   +37.348, E3 +423650.417}
SPL {X  -162.820, Y  +411.860, Z    +0.000, E1   +37.402, E3 +423663.568}
SPL {X  -162.820, Y  +407.726, Z    +0.000, E1   +37.291, E3 +423675.516}
SPL {X  -162.820, Y  +403.543, Z    +0.000, E1   +37.305, E3 +423686.862}
SPL {X  -162.820, Y  +399.300, Z    +0.000, E1   +37.355, E3 +423698.146}
SPL {X  -162.820, Y  +395.182, Z    +0.000, E1   +37.347, E3 +423709.435}
SPL {X  -162.820, Y  +390.797, Z    +0.000, E1   +37.358, E3 +423721.347}
SPL {X  -162.820, Y  +386.671, Z    +0.000, E1   +37.363, E3 +423732.528}
SPL {X  -162.820, Y  +382.174, Z    +0.000, E1   +37.329, E3 +423745.106}
SPL {X  -162.785, Y  +377.133, Z    +0.000, E1   +37.299, E3 +423759.035}
SPL {X  -162.623, Y  +372.484, Z    +0.000, E1   +37.337, E3 +423771.474}
SPL {X  -162.331, Y  +367.894, Z    +0.000, E1   +37.251, E3 +423784.587}
SPL {X  -161.920, Y  +363.407, Z    +0.000, E1   +37.164, E3 +423797.321}
SPL {X  -161.341, Y  +358.603, Z    +0.000, E1   +37.117, E3 +423810.801}
SPL {X  -160.616, Y  +353.801, Z    +0.000, E1   +36.942, E3 +423824.966}
SPL {X  -159.837, Y  +349.474, Z    +0.000, E1   +36.824, E3 +423837.410}
SPL {X  -159.171, Y  +346.224, Z    +0.000, E1   +36.747, E3 +423846.686}
SPL {X  -158.248, Y  +342.188, Z    +0.000, E1   +36.583, E3 +423858.849}
SPL {X  -153.520, Y  +326.260, Z    +0.000, E1   +41.363, E3 +423871.502}
SPL {X  -150.942, Y  +319.452, Z    +0.000, E1   +36.529, E3 +423927.859}
ENDSPLINE

SPLINE
SPL {X  -159.264, Y  +346.659, Z    +0.000, E1   +22.083, E3 +423968.433}
SPL {X  -161.245, Y  +357.907, Z    +0.000, E1   +16.095, E3 +423981.865}
SPL {X  -162.746, Y  +375.590, Z    +0.000, E1    +6.280, E3 +423981.454}
SPL {X  -162.820, Y  +384.478, Z    +0.000, E1    +0.434, E3 +423982.123}
SPL {X  -162.820, Y  +389.965, Z    +0.000, E1    -3.918, E3 +423981.835}
SPL {X  -162.820, Y  +394.532, Z    +0.000, E1    -7.849, E3 +423983.383}
SPL {X  -162.820, Y  +400.765, Z    +0.000, E1   -14.108, E3 +423980.850}
SPL {X  -162.820, Y  +411.829, Z    +0.000, E1   -24.195, E3 +423982.927}
SPL {X  -162.820, Y  +434.900, Z    +0.000, E1   -34.666, E3 +424010.292}
SPL {X  -162.820, Y  +465.440, Z    +0.000, E1   -41.264, E3 +424051.600}
ENDSPLINE

SPLINE
SPL {X  -162.820, Y  +460.175, Z    +0.000, E1   -36.098, E3 +424069.399}
ENDSPLINE

SPLINE
SPL {X  -162.820, Y  +467.031, Z    +0.000, E1   -36.178, E3 +424088.489}
SPL {X  -162.820, Y  +471.524, Z    +0.000, E1   -36.022, E3 +424102.042}
SPL {X  -162.820, Y  +475.701, Z    +0.000, E1   -36.157, E3 +424113.223}
SPL {X  -162.820, Y  +479.954, Z    +0.000, E1   -36.086, E3 +424125.764}
SPL {X  -162.820, Y  +483.976, Z    +0.000, E1   -36.049, E3 +424137.496}
SPL {X  -162.820, Y  +489.628, Z    +0.000, E1   -36.135, E3 +424153.326}
SPL {X  -162.820, Y  +494.712, Z    +0.000, E1   -36.164, E3 +424167.407}
SPL {X  -162.820, Y  +498.932, Z    +0.000, E1   -36.079, E3 +424180.134}
SPL {X  -162.820, Y  +504.528, Z    +0.000, E1   -36.109, E3 +424195.930}
SPL {X  -162.820, Y  +509.364, Z    +0.000, E1   -36.084, E3 +424209.835}
SPL {X  -162.820, Y  +515.001, Z    +0.000, E1   -36.183, E3 +424225.473}
SPL {X  -162.820, Y  +520.482, Z    +0.000, E1   -36.096, E3 +424241.519}
SPL {X  -162.820, Y  +524.107, Z    +0.000, E1   -36.045, E3 +424252.102}
SPL {X  -162.820, Y  +527.962, Z    +0.000, E1   -36.074, E3 +424263.035}
SPL {X  -162.820, Y  +532.253, Z    +0.000, E1   -36.170, E3 +424274.624}
SPL {X  -162.820, Y  +536.031, Z    +0.000, E1   -36.058, E3 +424286.162}
SPL {X  -162.820, Y  +541.179, Z    +0.000, E1   -36.085, E3 +424300.803}
SPL {X  -162.820, Y  +546.355, Z    +0.000, E1   -36.114, E3 +424315.347}
SPL {X  -162.820, Y  +550.585, Z    +0.000, E1   -36.077, E3 +424327.617}
SPL {X  -162.820, Y  +555.903, Z    +0.000, E1   -36.136, E3 +424342.615}
SPL {X  -162.820, Y  +561.684, Z    +0.000, E1   -36.118, E3 +424359.144}
SPL {X  -162.820, Y  +566.500, Z    +0.000, E1   -36.073, E3 +424373.147}
SPL {X  -162.820, Y  +570.319, Z    +0.000, E1   -36.045, E3 +424384.175}
SPL {X  -162.820, Y  +573.265, Z    +0.000, E1   -36.071, E3 +424392.411}
SPL {X  -162.820, Y  +576.887, Z    +0.000, E1   -36.084, E3 +424402.770}
SPL {X  -162.820, Y  +581.763, Z    +0.000, E1   -36.093, E3 +424416.707}
SPL {X  -162.820, Y  +586.693, Z    +0.000, E1   -36.086, E3 +424430.811}
SPL {X  -162.820, Y  +590.250, Z    +0.000, E1   -36.075, E3 +424440.930}
SPL {X  -162.820, Y  +592.727, Z    +0.000, E1   -35.960, E3 +424448.754}
SPL {X  -162.820, Y  +597.399, Z    +0.000, E1   -36.147, E3 +424461.103}
SPL {X  -162.820, Y  +602.243, Z    +0.000, E1   -36.085, E3 +424475.249}
SPL {X  -162.820, Y  +605.848, Z    +0.000, E1   -36.070, E3 +424485.570}
SPL {X  -162.820, Y  +609.375, Z    +0.000, E1   -36.084, E3 +424495.620}
SPL {X  -162.820, Y  +612.959, Z    +0.000, E1   -36.034, E3 +424506.140}
SPL {X  -162.820, Y  +616.897, Z    +0.000, E1   -36.061, E3 +424517.288}
SPL {X  -162.820, Y  +620.590, Z    +0.000, E1   -36.079, E3 +424527.683}
SPL {X  -162.820, Y  +625.276, Z    +0.000, E1   -36.104, E3 +424541.100}
SPL {X  -162.820, Y  +630.571, Z    +0.000, E1   -36.057, E3 +424556.432}
SPL {X  -162.820, Y  +634.189, Z    +0.000, E1   -36.065, E3 +424566.625}
SPL {X  -162.820, Y  +638.473, Z    +0.000, E1   -36.098, E3 +424578.862}
SPL {X  -162.820, Y  +642.832, Z    +0.000, E1   -36.091, E3 +424591.188}
SPL {X  -162.820, Y  +646.320, Z    +0.000, E1   -36.078, E3 +424601.295}
SPL {X  -162.820, Y  +651.289, Z    +0.000, E1   -36.059, E3 +424615.752}
SPL {X  -162.820, Y  +656.677, Z    +0.000, E1   -36.110, E3 +424630.765}
SPL {X  -162.820, Y  +661.560, Z    +0.000, E1   -36.068, E3 +424645.028}
SPL {X  -162.820, Y  +666.386, Z    +0.000, E1   -36.048, E3 +424658.912}
SPL {X  -162.820, Y  +671.104, Z    +0.000, E1   -36.061, E3 +424672.332}
SPL {X  -162.787, Y  +676.764, Z    +0.000, E1   -36.126, E3 +424688.231}
SPL {X  -162.633, Y  +681.311, Z    +0.000, E1   -35.984, E3 +424701.920}
SPL {X  -162.367, Y  +685.641, Z    +0.000, E1   -36.000, E3 +424714.328}
SPL {X  -161.948, Y  +690.331, Z    +0.000, E1   -35.960, E3 +424727.923}
SPL {X  -161.544, Y  +693.846, Z    +0.000, E1   -35.908, E3 +424738.198}
SPL {X  -160.925, Y  +698.267, Z    +0.000, E1   -35.816, E3 +424751.630}
SPL {X  -160.151, Y  +702.861, Z    +0.000, E1   -35.643, E3 +424765.600}
SPL {X  -159.622, Y  +705.613, Z    +0.000, E1   -35.430, E3 +424774.719}
SPL {X  -158.758, Y  +709.640, Z    +0.000, E1   -35.380, E3 +424786.726}
SPL {X  -155.037, Y  +723.239, Z    +0.000, E1   -39.382, E3 +424799.611}
SPL {X  -152.141, Y  +731.494, Z    +0.000, E1   -35.181, E3 +424858.417}
ENDSPLINE

SPLINE
SPL {X  -160.133, Y  +702.956, Z    +0.000, E1   -19.806, E3 +424901.955}
SPL {X  -161.979, Y  +690.023, Z    +0.000, E1   -12.991, E3 +424904.872}
SPL {X  -162.641, Y  +681.139, Z    +0.000, E1    -7.893, E3 +424906.963}
SPL {X  -162.820, Y  +673.062, Z    +0.000, E1    -2.992, E3 +424905.930}
SPL {X  -162.820, Y  +666.731, Z    +0.000, E1    +1.545, E3 +424907.560}
SPL {X  -162.820, Y  +660.758, Z    +0.000, E1    +6.523, E3 +424907.271}
SPL {X  -162.820, Y  +650.583, Z    +0.000, E1   +16.035, E3 +424906.243}
SPL {X  -162.820, Y  +629.267, Z    +0.000, E1   +31.872, E3 +424917.392}
SPL {X  -162.820, Y  +617.390, Z    +0.000, E1   +35.413, E3 +424934.321}
SPL {X  -162.820, Y  +596.392, Z    +0.000, E1   +37.895, E3 +424975.061}
ENDSPLINE

SPLINE
SPL {X  -162.820, Y  +599.924, Z    +0.000, E1   +33.992, E3 +424989.435}
ENDSPLINE

SPLINE
SPL {X  -162.820, Y  +595.170, Z    +0.000, E1   +33.784, E3 +425005.483}
SPL {X  -162.820, Y  +589.785, Z    +0.000, E1   +33.904, E3 +425021.480}
SPL {X  -162.820, Y  +584.646, Z    +0.000, E1   +33.882, E3 +425037.550}
SPL {X  -162.820, Y  +579.919, Z    +0.000, E1   +33.857, E3 +425052.338}
SPL {X  -162.820, Y  +574.615, Z    +0.000, E1   +33.920, E3 +425068.512}
SPL {X  -162.820, Y  +570.335, Z    +0.000, E1   +33.821, E3 +425082.217}
SPL {X  -162.820, Y  +565.901, Z    +0.000, E1   +33.889, E3 +425095.738}
SPL {X  -162.820, Y  +562.173, Z    +0.000, E1   +33.897, E3 +425107.029}
SPL {X  -162.820, Y  +559.395, Z    +0.000, E1   +33.796, E3 +425116.396}
SPL {X  -162.820, Y  +554.453, Z    +0.000, E1   +33.841, E3 +425131.620}
SPL {X  -162.820, Y  +549.726, Z    +0.000, E1   +33.905, E3 +425145.724}
SPL {X  -162.820, Y  +545.760, Z    +0.000, E1   +33.901, E3 +425158.120}
SPL {X  -162.820, Y  +541.668, Z    +0.000, E1   +33.787, E3 +425171.520}
SPL {X  -162.820, Y  +537.061, Z    +0.000, E1   +33.897, E3 +425185.178}
SPL {X  -162.820, Y  +532.164, Z    +0.000, E1   +33.861, E3 +425200.652}
SPL {X  -162.820, Y  +528.475, Z    +0.000, E1   +33.876, E3 +425211.821}
SPL {X  -162.820, Y  +524.900, Z    +0.000, E1   +33.820, E3 +425223.479}
SPL {X  -162.820, Y  +520.532, Z    +0.000, E1   +33.805, E3 +425237.047}
SPL {X  -162.820, Y  +516.814, Z    +0.000, E1   +33.917, E3 +425247.883}
SPL {X  -162.820, Y  +512.685, Z    +0.000, E1   +33.830, E3 +425261.326}
SPL {X  -162.820, Y  +508.888, Z    +0.000, E1   +33.871, E3 +425272.741}
SPL {X  -162.820, Y  +505.651, Z    +0.000, E1   +33.839, E3 +425283.058}
SPL {X  -162.820, Y  +500.931, Z    +0.000, E1   +34.256, E3 +425294.931}
SPL {X  -162.820, Y  +481.122, Z    +0.000, E1   +41.279, E3 +425305.196}
SPL {X  -162.820, Y  +477.698, Z    +0.000, E1   +40.353, E3 +425319.252}
SPL {X  -162.820, Y  +474.538, Z    +0.000, E1   +39.267, E3 +425333.427}
SPL {X  -162.820, Y  +472.097, Z    +0.000, E1   +38.411, E3 +425344.971}
SPL {X  -162.820, Y  +469.308, Z    +0.000, E1   +37.839, E3 +425355.775}
SPL {X  -162.820, Y  +467.216, Z    +0.000, E1   +37.215, E3 +425365.341}
SPL {X  -162.820, Y  +462.598, Z    +0.000, E1   +37.325, E3 +425377.295}
SPL {X  -162.820, Y  +457.832, Z    +0.000, E1   +37.294, E3 +425390.582}
SPL {X  -162.820, Y  +452.986, Z    +0.000, E1   +37.368, E3 +425403.316}
SPL {X  -162.820, Y  +448.311, Z    +0.000, E1   +37.333, E3 +425416.336}
SPL {X  -162.820, Y  +443.351, Z    +0.000, E1   +37.335, E3 +425429.866}
SPL {X  -162.820, Y  +438.727, Z    +0.000, E1   +37.289, E3 +425442.738}
SPL {X  -162.820, Y  +434.320, Z    +0.000, E1   +37.343, E3 +425454.448}
SPL {X  -162.820, Y  +430.091, Z    +0.000, E1   +37.424, E3 +425465.448}
SPL {X  -162.820, Y  +426.177, Z    +0.000, E1   +37.250, E3 +425477.271}
SPL {X  -162.820, Y  +421.391, Z    +0.000, E1   +37.346, E3 +425489.734}
SPL {X  -162.820, Y  +416.811, Z    +0.000, E1   +37.348, E3 +425502.269}
SPL {X  -162.820, Y  +411.860, Z    +0.000, E1   +37.402, E3 +425515.420}
SPL {X  -162.820, Y  +407.726, Z    +0.000, E1   +37.291, E3 +425527.368}
SPL {X  -162.820, Y  +403.543, Z    +0.000, E1   +37.305, E3 +425538.714}
SPL {X  -162.820, Y  +399.300, Z    +0.000, E1   +37.355, E3 +425549.998}
SPL {X  -162.820, Y  +395.182, Z    +0.000, E1   +37.347, E3 +425561.287}
SPL {X  -162.820, Y  +390.797, Z    +0.000, E1   +37.358, E3 +425573.199}
SPL {X  -162.820, Y  +386.671, Z    +0.000, E1   +37.363, E3 +425584.380}
SPL {X  -162.820, Y  +382.174, Z    +0.000, E1   +37.329, E3 +425596.957}
SPL {X  -162.785, Y  +377.133, Z    +0.000, E1   +37.299, E3 +425610.887}
SPL {X  -162.576, Y  +371.586, Z    +0.000, E1   +37.322, E3 +425625.999}
SPL {X  -162.256, Y  +366.963, Z    +0.000, E1   +37.251, E3 +425638.888}
SPL {X  -161.920, Y  +363.407, Z    +0.000, E1   +37.164, E3 +425649.173}
SPL {X  -161.341, Y  +358.603, Z    +0.000, E1   +37.117, E3 +425662.653}
SPL {X  -160.616, Y  +353.801, Z    +0.000, E1   +36.942, E3 +425676.818}
SPL {X  -159.837, Y  +349.474, Z    +0.000, E1   +36.824, E3 +425689.262}
SPL {X  -158.862, Y  +344.820, Z    +0.000, E1   +36.732, E3 +425702.624}
SPL {X  -157.959, Y  +341.011, Z    +0.000, E1   +36.448, E3 +425714.521}
SPL {X  -153.520, Y  +326.260, Z    +0.000, E1   +41.363, E3 +425723.353}
SPL {X  -150.942, Y  +319.452, Z    +0.000, E1   +36.529, E3 +425779.710}
ENDSPLINE

SPLINE
SPL {X  -159.264, Y  +346.659, Z    +0.000, E1   +22.083, E3 +425820.285}
SPL {X  -161.245, Y  +357.907, Z    +0.000, E1   +16.095, E3 +425833.717}
SPL {X  -162.697, Y  +374.161, Z    +0.000, E1    +7.119, E3 +425831.707}
SPL {X  -162.820, Y  +380.878, Z    +0.000, E1    +2.854, E3 +425834.538}
SPL {X  -162.820, Y  +385.313, Z    +0.000, E1    -0.228, E3 +425834.318}
SPL {X  -162.820, Y  +389.965, Z    +0.000, E1    -3.918, E3 +425833.687}
SPL {X  -162.820, Y  +394.532, Z    +0.000, E1    -7.849, E3 +425835.235}
SPL {X  -162.820, Y  +400.765, Z    +0.000, E1   -14.108, E3 +425832.702}
SPL {X  -162.820, Y  +411.829, Z    +0.000, E1   -24.195, E3 +425834.779}
SPL {X  -162.820, Y  +434.900, Z    +0.000, E1   -34.666, E3 +425862.144}
SPL {X  -162.820, Y  +465.440, Z    +0.000, E1   -41.264, E3 +425903.451}
ENDSPLINE

SPLINE
SPL {X  -162.820, Y  +460.175, Z    +0.000, E1   -36.098, E3 +425921.251}
ENDSPLINE

SPLINE
SPL {X  -162.820, Y  +465.690, Z    +0.000, E1   -36.140, E3 +425936.565}
SPL {X  -162.820, Y  +470.432, Z    +0.000, E1   -36.100, E3 +425950.448}
SPL {X  -162.820, Y  +475.701, Z    +0.000, E1   -36.157, E3 +425965.075}
SPL {X  -162.820, Y  +479.954, Z    +0.000, E1   -36.086, E3 +425977.616}
SPL {X  -162.820, Y  +485.438, Z    +0.000, E1   -36.112, E3 +425993.334}
SPL {X  -162.820, Y  +490.843, Z    +0.000, E1   -36.087, E3 +426008.747}
SPL {X  -162.820, Y  +494.712, Z    +0.000, E1   -36.164, E3 +426019.259}
SPL {X  -162.820, Y  +498.932, Z    +0.000, E1   -36.079, E3 +426031.986}
SPL {X  -162.820, Y  +504.528, Z    +0.000, E1   -36.109, E3 +426047.782}
SPL {X  -162.820, Y  +509.364, Z    +0.000, E1   -36.084, E3 +426061.687}
SPL {X  -162.820, Y  +515.001, Z    +0.000, E1   -36.183, E3 +426077.325}
SPL {X  -162.820, Y  +520.482, Z    +0.000, E1   -36.096, E3 +426093.370}
SPL {X  -162.820, Y  +524.107, Z    +0.000, E1   -36.045, E3 +426103.954}
SPL {X  -162.820, Y  +527.962, Z    +0.000, E1   -36.074, E3 +426114.887}
SPL {X  -162.820, Y  +532.253, Z    +0.000, E1   -36.170, E3 +426126.476}
SPL {X  -162.820, Y  +536.031, Z    +0.000, E1   -36.058, E3 +426138.014}
SPL {X  -162.820, Y  +541.179, Z    +0.000, E1   -36.085, E3 +426152.655}
SPL {X  -162.820, Y  +546.355, Z    +0.000, E1   -36.114, E3 +426167.199}
SPL {X  -162.820, Y  +551.776, Z    +0.000, E1   -36.108, E3 +426182.833}
SPL {X  -162.820, Y  +556.944, Z    +0.000, E1   -36.118, E3 +426197.404}
SPL {X  -162.820, Y  +561.684, Z    +0.000, E1   -36.118, E3 +426210.996}
SPL {X  -162.820, Y  +566.500, Z    +0.000, E1   -36.073, E3 +426224.999}
SPL {X  -162.820, Y  +571.734, Z    +0.000, E1   -36.094, E3 +426239.928}
SPL {X  -162.820, Y  +576.887, Z    +0.000, E1   -36.084, E3 +426254.622}
SPL {X  -162.820, Y  +581.763, Z    +0.000, E1   -36.093, E3 +426268.558}
SPL {X  -162.820, Y  +586.693, Z    +0.000, E1   -36.086, E3 +426282.663}
SPL {X  -162.820, Y  +590.250, Z    +0.000, E1   -36.075, E3 +426292.782}
SPL {X  -162.820, Y  +592.727, Z    +0.000, E1   -35.960, E3 +426300.606}
SPL {X  -162.820, Y  +597.399, Z    +0.000, E1   -36.147, E3 +426312.954}
SPL {X  -162.820, Y  +602.243, Z    +0.000, E1   -36.085, E3 +426327.101}
SPL {X  -162.820, Y  +606.975, Z    +0.000, E1   -36.102, E3 +426340.546}
SPL {X  -162.820, Y  +611.980, Z    +0.000, E1   -36.072, E3 +426355.091}
SPL {X  -162.820, Y  +616.897, Z    +0.000, E1   -36.061, E3 +426369.140}
SPL {X  -162.820, Y  +621.516, Z    +0.000, E1   -36.072, E3 +426382.339}
SPL {X  -162.820, Y  +626.243, Z    +0.000, E1   -36.105, E3 +426395.582}
SPL {X  -162.820, Y  +630.571, Z    +0.000, E1   -36.057, E3 +426408.284}
SPL {X  -162.820, Y  +634.189, Z    +0.000, E1   -36.065, E3 +426418.477}
SPL {X  -162.820, Y  +638.473, Z    +0.000, E1   -36.098, E3 +426430.714}
SPL {X  -162.820, Y  +642.832, Z    +0.000, E1   -36.091, E3 +426443.040}
SPL {X  -162.820, Y  +646.320, Z    +0.000, E1   -36.078, E3 +426453.147}
SPL {X  -162.820, Y  +651.289, Z    +0.000, E1   -36.059, E3 +426467.604}
SPL {X  -162.820, Y  +656.677, Z    +0.000, E1   -36.110, E3 +426482.617}
SPL {X  -162.820, Y  +660.489, Z    +0.000, E1   -36.068, E3 +426493.683}
SPL {X  -162.820, Y  +665.459, Z    +0.000, E1   -36.068, E3 +426508.130}
SPL {X  -162.820, Y  +669.858, Z    +0.000, E1   -36.039, E3 +426520.641}
SPL {X  -162.820, Y  +673.415, Z    +0.000, E1   -36.053, E3 +426530.851}
SPL {X  -162.761, Y  +677.889, Z    +0.000, E1   -36.122, E3 +426543.169}
SPL {X  -162.633, Y  +681.311, Z    +0.000, E1   -35.984, E3 +426553.772}
SPL {X  -162.367, Y  +685.641, Z    +0.000, E1   -36.000, E3 +426566.180}
SPL {X  -161.948, Y  +690.331, Z    +0.000, E1   -35.960, E3 +426579.775}
SPL {X  -161.544, Y  +693.846, Z    +0.000, E1   -35.908, E3 +426590.050}
SPL {X  -161.078, Y  +697.256, Z    +0.000, E1   -35.797, E3 +426600.556}
SPL {X  -160.313, Y  +701.964, Z    +0.000, E1   -35.709, E3 +426614.632}
SPL {X  -159.622, Y  +705.613, Z    +0.000, E1   -35.430, E3 +426626.571}
SPL {X  -158.758, Y  +709.640, Z    +0.000, E1   -35.380, E3 +426638.578}
SPL {X  -155.037, Y  +723.239, Z    +0.000, E1   -39.382, E3 +426651.463}
SPL {X  -152.141, Y  +731.494, Z    +0.000, E1   -35.181, E3 +426710.269}
ENDSPLINE

SPLINE
SPL {X  -160.133, Y  +702.956, Z    +0.000, E1   -19.806, E3 +426753.807}
SPL {X  -161.979, Y  +690.023, Z    +0.000, E1   -12.991, E3 +426756.724}
SPL {X  -162.641, Y  +681.139, Z    +0.000, E1    -7.893, E3 +426758.815}
SPL {X  -162.820, Y  +673.062, Z    +0.000, E1    -2.992, E3 +426757.782}
SPL {X  -162.820, Y  +666.731, Z    +0.000, E1    +1.545, E3 +426759.412}
SPL {X  -162.820, Y  +660.758, Z    +0.000, E1    +6.523, E3 +426759.123}
SPL {X  -162.820, Y  +650.583, Z    +0.000, E1   +16.035, E3 +426758.095}
SPL {X  -162.820, Y  +629.267, Z    +0.000, E1   +31.872, E3 +426769.244}
SPL {X  -162.820, Y  +620.680, Z    +0.000, E1   +34.107, E3 +426783.293}
SPL {X  -162.820, Y  +609.002, Z    +0.000, E1   +38.458, E3 +426793.444}
SPL {X  -162.820, Y  +596.392, Z    +0.000, E1   +37.895, E3 +426826.913}
ENDSPLINE

SPLINE
SPL {X  -162.820, Y  +599.924, Z    +0.000, E1   +33.992, E3 +426841.287}
ENDSPLINE

SPLINE
SPL {X  -162.820, Y  +595.170, Z    +0.000, E1   +33.784, E3 +426857.335}
SPL {X  -162.820, Y  +589.785, Z    +0.000, E1   +33.904, E3 +426873.332}
SPL {X  -162.820, Y  +584.646, Z    +0.000, E1   +33.882, E3 +426889.401}
SPL {X  -162.820, Y  +579.919, Z    +0.000, E1   +33.857, E3 +426904.189}
SPL {X  -162.820, Y  +574.615, Z    +0.000, E1   +33.920, E3 +426920.363}
SPL {X  -162.820, Y  +570.335, Z    +0.000, E1   +33.821, E3 +426934.069}
SPL {X  -162.820, Y  +565.901, Z    +0.000, E1   +33.889, E3 +426947.589}
SPL {X  -162.820, Y  +560.226, Z    +0.000, E1   +33.868, E3 +426965.375}
SPL {X  -162.820, Y  +554.453, Z    +0.000, E1   +33.841, E3 +426983.472}
SPL {X  -162.820, Y  +549.726, Z    +0.000, E1   +33.905, E3 +426997.576}
SPL {X  -162.820, Y  +545.760, Z    +0.000, E1   +33.901, E3 +427009.972}
SPL {X  -162.820, Y  +541.668, Z    +0.000, E1   +33.787, E3 +427023.372}
SPL {X  -162.820, Y  +538.174, Z    +0.000, E1   +33.865, E3 +427033.661}
SPL {X  -162.820, Y  +534.943, Z    +0.000, E1   +33.919, E3 +427043.401}
SPL {X  -162.820, Y  +530.273, Z    +0.000, E1   +33.855, E3 +427058.431}
SPL {X  -162.820, Y  +524.900, Z    +0.000, E1   +33.820, E3 +427075.331}
SPL {X  -162.820, Y  +520.532, Z    +0.000, E1   +33.805, E3 +427088.899}
SPL {X  -162.820, Y  +516.814, Z    +0.000, E1   +33.917, E3 +427099.735}
SPL {X  -162.820, Y  +512.685, Z    +0.000, E1   +33.830, E3 +427113.178}
SPL {X  -162.820, Y  +508.888, Z    +0.000, E1   +33.871, E3 +427124.592}
SPL {X  -162.820, Y  +505.651, Z    +0.000, E1   +33.839, E3 +427134.909}
SPL {X  -162.820, Y  +500.931, Z    +0.000, E1   +34.256, E3 +427146.783}
SPL {X  -162.820, Y  +481.122, Z    +0.000, E1   +41.279, E3 +427157.047}
SPL {X  -162.820, Y  +478.698, Z    +0.000, E1   +40.526, E3 +427167.396}
SPL {X  -162.820, Y  +475.203, Z    +0.000, E1   +39.596, E3 +427181.856}
SPL {X  -162.820, Y  +472.097, Z    +0.000, E1   +38.411, E3 +427196.823}
SPL {X  -162.820, Y  +469.308, Z    +0.000, E1   +37.839, E3 +427207.627}
SPL {X  -162.820, Y  +467.216, Z    +0.000, E1   +37.215, E3 +427217.193}
SPL {X  -162.820, Y  +462.598, Z    +0.000, E1   +37.325, E3 +427229.147}
SPL {X  -162.820, Y  +457.832, Z    +0.000, E1   +37.294, E3 +427242.434}
SPL {X  -162.820, Y  +452.986, Z    +0.000, E1   +37.368, E3 +427255.168}
SPL {X  -162.820, Y  +448.311, Z    +0.000, E1   +37.333, E3 +427268.188}
SPL {X  -162.820, Y  +443.351, Z    +0.000, E1   +37.335, E3 +427281.717}
SPL {X  -162.820, Y  +438.727, Z    +0.000, E1   +37.289, E3 +427294.590}
SPL {X  -162.820, Y  +434.320, Z    +0.000, E1   +37.343, E3 +427306.300}
SPL {X  -162.820, Y  +430.091, Z    +0.000, E1   +37.424, E3 +427317.300}
SPL {X  -162.820, Y  +426.177, Z    +0.000, E1   +37.250, E3 +427329.123}
SPL {X  -162.820, Y  +420.241, Z    +0.000, E1   +37.355, E3 +427344.829}
SPL {X  -162.820, Y  +415.595, Z    +0.000, E1   +37.375, E3 +427357.169}
SPL {X  -162.820, Y  +411.860, Z    +0.000, E1   +37.402, E3 +427367.272}
SPL {X  -162.820, Y  +407.726, Z    +0.000, E1   +37.291, E3 +427379.220}
SPL {X  -162.820, Y  +403.543, Z    +0.000, E1   +37.305, E3 +427390.565}
SPL {X  -162.820, Y  +399.300, Z    +0.000, E1   +37.355, E3 +427401.850}
SPL {X  -162.820, Y  +395.182, Z    +0.000, E1   +37.347, E3 +427413.139}
SPL {X  -162.820, Y  +390.797, Z    +0.000, E1   +37.358, E3 +427425.051}
SPL {X  -162.820, Y  +386.671, Z    +0.000, E1   +37.363, E3 +427436.232}
SPL {X  -162.820, Y  +382.174, Z    +0.000, E1   +37.329, E3 +427448.809}
SPL {X  -162.785, Y  +377.133, Z    +0.000, E1   +37.299, E3 +427462.738}
SPL {X  -162.623, Y  +372.484, Z    +0.000, E1   +37.337, E3 +427475.178}
SPL {X  -162.331, Y  +367.894, Z    +0.000, E1   +37.251, E3 +427488.291}
SPL {X  -161.920, Y  +363.407, Z    +0.000, E1   +37.164, E3 +427501.025}
SPL {X  -161.482, Y  +359.669, Z    +0.000, E1   +37.064, E3 +427511.810}
SPL {X  -160.943, Y  +355.851, Z    +0.000, E1   +37.136, E3 +427521.796}
SPL {X  -160.493, Y  +353.069, Z    +0.000, E1   +36.789, E3 +427531.448}
SPL {X  -159.837, Y  +349.474, Z    +0.000, E1   +36.824, E3 +427541.114}
SPL {X  -159.171, Y  +346.224, Z    +0.000, E1   +36.747, E3 +427550.390}
SPL {X  -158.248, Y  +342.188, Z    +0.000, E1   +36.583, E3 +427562.553}
SPL {X  -153.520, Y  +326.260, Z    +0.000, E1   +41.363, E3 +427575.205}
SPL {X  -150.942, Y  +319.452, Z    +0.000, E1   +36.529, E3 +427631.562}
ENDSPLINE

SPLINE
SPL {X  -159.264, Y  +346.659, Z    +0.000, E1   +22.083, E3 +427672.136}
SPL {X  -161.245, Y  +357.907, Z    +0.000, E1   +16.095, E3 +427685.569}
SPL {X  -162.746, Y  +375.590, Z    +0.000, E1    +6.280, E3 +427685.158}
SPL {X  -162.820, Y  +384.478, Z    +0.000, E1    +0.434, E3 +427685.827}
SPL {X  -162.820, Y  +389.965, Z    +0.000, E1    -3.918, E3 +427685.539}
SPL {X  -162.820, Y  +394.532, Z    +0.000, E1    -7.849, E3 +427687.087}
SPL {X  -162.820, Y  +400.765, Z    +0.000, E1   -14.108, E3 +427684.554}
SPL {X  -162.820, Y  +411.829, Z    +0.000, E1   -24.195, E3 +427686.631}
SPL {X  -162.820, Y  +434.900, Z    +0.000, E1   -34.666, E3 +427713.996}
SPL {X  -162.820, Y  +465.440, Z    +0.000, E1   -41.264, E3 +427755.303}
ENDSPLINE

SPLINE
SPL {X  -162.820, Y  +460.175, Z    +0.000, E1   -36.098, E3 +427773.103}
ENDSPLINE

SPLINE
SPL {X  -162.820, Y  +467.031, Z    +0.000, E1   -36.178, E3 +427792.193}
SPL {X  -162.820, Y  +471.524, Z    +0.000, E1   -36.022, E3 +427805.746}
SPL {X  -162.820, Y  +475.701, Z    +0.000, E1   -36.157, E3 +427816.927}
SPL {X  -162.820, Y  +479.954, Z    +0.000, E1   -36.086, E3 +427829.468}
SPL {X  -162.820, Y  +485.438, Z    +0.000, E1   -36.112, E3 +427845.186}
SPL {X  -162.820, Y  +490.843, Z    +0.000, E1   -36.087, E3 +427860.599}
SPL {X  -162.820, Y  +494.712, Z    +0.000, E1   -36.164, E3 +427871.111}
SPL {X  -162.820, Y  +497.796, Z    +0.000, E1   -36.022, E3 +427880.817}
SPL {X  -162.820, Y  +502.146, Z    +0.000, E1   -36.123, E3 +427892.686}
SPL {X  -162.820, Y  +505.688, Z    +0.000, E1   -36.050, E3 +427903.168}
SPL {X  -162.820, Y  +509.364, Z    +0.000, E1   -36.084, E3 +427913.539}
SPL {X  -162.820, Y  +513.393, Z    +0.000, E1   -36.179, E3 +427924.395}
SPL {X  -162.820, Y  +516.436, Z    +0.000, E1   -36.094, E3 +427933.591}
SPL {X  -162.820, Y  +520.482, Z    +0.000, E1   -36.096, E3 +427945.222}
SPL {X  -162.820, Y  +524.107, Z    +0.000, E1   -36.045, E3 +427955.806}
SPL {X  -162.820, Y  +527.962, Z    +0.000, E1   -36.074, E3 +427966.739}
SPL {X  -162.820, Y  +532.253, Z    +0.000, E1   -36.170, E3 +427978.328}
SPL {X  -162.820, Y  +536.031, Z    +0.000, E1   -36.058, E3 +427989.866}
SPL {X  -162.820, Y  +541.179, Z    +0.000, E1   -36.085, E3 +428004.507}
SPL {X  -162.820, Y  +546.355, Z    +0.000, E1   -36.114, E3 +428019.051}
SPL {X  -162.820, Y  +551.776, Z    +0.000, E1   -36.108, E3 +428034.685}
SPL {X  -162.820, Y  +558.272, Z    +0.000, E1   -36.170, E3 +428052.893}
SPL {X  -162.820, Y  +562.721, Z    +0.000, E1   -36.046, E3 +428066.118}
SPL {X  -162.820, Y  +566.500, Z    +0.000, E1   -36.073, E3 +428076.850}
SPL {X  -162.820, Y  +570.319, Z    +0.000, E1   -36.045, E3 +428087.878}
SPL {X  -162.820, Y  +573.265, Z    +0.000, E1   -36.071, E3 +428096.115}
SPL {X  -162.820, Y  +576.887, Z    +0.000, E1   -36.084, E3 +428106.473}
SPL {X  -162.820, Y  +581.763, Z    +0.000, E1   -36.093, E3 +428120.410}
SPL {X  -162.820, Y  +586.693, Z    +0.000, E1   -36.086, E3 +428134.515}
SPL {X  -162.820, Y  +591.665, Z    +0.000, E1   -36.045, E3 +428149.043}
SPL {X  -162.820, Y  +597.399, Z    +0.000, E1   -36.147, E3 +428164.806}
SPL {X  -162.820, Y  +602.243, Z    +0.000, E1   -36.085, E3 +428178.952}
SPL {X  -162.820, Y  +605.848, Z    +0.000, E1   -36.070, E3 +428189.274}
SPL {X  -162.820, Y  +609.375, Z    +0.000, E1   -36.084, E3 +428199.324}
SPL {X  -162.820, Y  +612.959, Z    +0.000, E1   -36.034, E3 +428209.844}
SPL {X  -162.820, Y  +616.897, Z    +0.000, E1   -36.061, E3 +428220.992}
SPL {X  -162.820, Y  +621.516, Z    +0.000, E1   -36.072, E3 +428234.191}
SPL {X  -162.820, Y  +626.243, Z    +0.000, E1   -36.105, E3 +428247.434}
SPL {X  -162.820, Y  +630.571, Z    +0.000, E1   -36.057, E3 +428260.136}
SPL {X  -162.820, Y  +634.189, Z    +0.000, E1   -36.065, E3 +428270.329}
SPL {X  -162.820, Y  +638.473, Z    +0.000, E1   -36.098, E3 +428282.566}
SPL {X  -162.820, Y  +642.832, Z    +0.000, E1   -36.091, E3 +428294.892}
SPL {X  -162.820, Y  +646.320, Z    +0.000, E1   -36.078, E3 +428304.999}
SPL {X  -162.820, Y  +651.289, Z    +0.000, E1   -36.059, E3 +428319.456}
SPL {X  -162.820, Y  +656.677, Z    +0.000, E1   -36.110, E3 +428334.469}
SPL {X  -162.820, Y  +661.560, Z    +0.000, E1   -36.068, E3 +428348.732}
SPL {X  -162.820, Y  +666.386, Z    +0.000, E1   -36.048, E3 +428362.616}
SPL {X  -162.820, Y  +671.104, Z    +0.000, E1   -36.061, E3 +428376.036}
SPL {X  -162.787, Y  +676.764, Z    +0.000, E1   -36.126, E3 +428391.935}
SPL {X  -162.633, Y  +681.311, Z    +0.000, E1   -35.984, E3 +428405.624}
SPL {X  -162.367, Y  +685.641, Z    +0.000, E1   -36.000, E3 +428418.031}
SPL {X  -162.041, Y  +689.412, Z    +0.000, E1   -36.001, E3 +428428.651}
SPL {X  -161.667, Y  +692.839, Z    +0.000, E1   -35.918, E3 +428439.072}
SPL {X  -161.078, Y  +697.256, Z    +0.000, E1   -35.797, E3 +428452.408}
SPL {X  -160.313, Y  +701.964, Z    +0.000, E1   -35.709, E3 +428466.484}
SPL {X  -159.622, Y  +705.613, Z    +0.000, E1   -35.430, E3 +428478.423}
SPL {X  -158.758, Y  +709.640, Z    +0.000, E1   -35.380, E3 +428490.430}
SPL {X  -155.037, Y  +723.239, Z    +0.000, E1   -39.382, E3 +428503.315}
SPL {X  -152.141, Y  +731.494, Z    +0.000, E1   -35.181, E3 +428562.121}
ENDSPLINE

SPLINE
SPL {X  -160.133, Y  +702.956, Z    +0.000, E1   -19.806, E3 +428605.659}
SPL {X  -161.979, Y  +690.023, Z    +0.000, E1   -12.991, E3 +428608.575}
SPL {X  -162.641, Y  +681.139, Z    +0.000, E1    -7.893, E3 +428610.667}
SPL {X  -162.820, Y  +673.062, Z    +0.000, E1    -2.992, E3 +428609.634}
SPL {X  -162.820, Y  +665.516, Z    +0.000, E1    +2.410, E3 +428611.474}
SPL {X  -162.820, Y  +657.781, Z    +0.000, E1    +9.391, E3 +428609.138}
SPL {X  -162.820, Y  +648.706, Z    +0.000, E1   +17.761, E3 +428610.890}
SPL {X  -162.820, Y  +629.267, Z    +0.000, E1   +31.872, E3 +428621.096}
SPL {X  -162.820, Y  +617.390, Z    +0.000, E1   +35.413, E3 +428638.025}
SPL {X  -162.820, Y  +596.392, Z    +0.000, E1   +37.895, E3 +428678.765}
ENDSPLINE

SPLINE
SPL {X  -162.820, Y  +599.924, Z    +0.000, E1   +33.992, E3 +428693.139}
ENDSPLINE

SPLINE
SPL {X  -162.820, Y  +596.128, Z    +0.000, E1   +33.827, E3 +428705.777}
SPL {X  -162.820, Y  +592.692, Z    +0.000, E1   +33.779, E3 +428716.852}
SPL {X  -162.820, Y  +588.795, Z    +0.000, E1   +33.876, E3 +428728.289}
SPL {X  -162.820, Y  +585.519, Z    +0.000, E1   +33.888, E3 +428738.374}
SPL {X  -162.820, Y  +582.066, Z    +0.000, E1   +33.857, E3 +428749.308}
SPL {X  -162.820, Y  +577.919, Z    +0.000, E1   +33.841, E3 +428762.361}
SPL {X  -162.820, Y  +573.566, Z    +0.000, E1   +33.899, E3 +428775.436}
SPL {X  -162.820, Y  +569.298, Z    +0.000, E1   +33.851, E3 +428789.077}
SPL {X  -162.820, Y  +565.024, Z    +0.000, E1   +33.872, E3 +428802.133}
SPL {X  -162.820, Y  +560.226, Z    +0.000, E1   +33.868, E3 +428817.227}
SPL {X  -162.820, Y  +556.206, Z    +0.000, E1   +33.843, E3 +428829.627}
SPL {X  -162.820, Y  +553.486, Z    +0.000, E1   +33.777, E3 +428838.573}
SPL {X  -162.820, Y  +548.576, Z    +0.000, E1   +33.950, E3 +428852.854}
SPL {X  -162.820, Y  +544.808, Z    +0.000, E1   +33.827, E3 +428865.117}
SPL {X  -162.820, Y  +541.668, Z    +0.000, E1   +33.787, E3 +428875.223}
SPL {X  -162.820, Y  +538.174, Z    +0.000, E1   +33.865, E3 +428885.513}
SPL {X  -162.820, Y  +534.943, Z    +0.000, E1   +33.919, E3 +428895.253}
SPL {X  -162.820, Y  +531.459, Z    +0.000, E1   +33.783, E3 +428906.910}
SPL {X  -162.820, Y  +528.475, Z    +0.000, E1   +33.876, E3 +428915.524}
SPL {X  -162.820, Y  +524.900, Z    +0.000, E1   +33.820, E3 +428927.183}
SPL {X  -162.820, Y  +520.532, Z    +0.000, E1   +33.805, E3 +428940.751}
SPL {X  -162.820, Y  +515.754, Z    +0.000, E1   +33.911, E3 +428955.087}
SPL {X  -162.820, Y  +510.207, Z    +0.000, E1   +33.879, E3 +428972.467}
SPL {X  -162.820, Y  +505.651, Z    +0.000, E1   +33.839, E3 +428986.761}
SPL {X  -162.820, Y  +500.931, Z    +0.000, E1   +34.256, E3 +428998.635}
SPL {X  -162.820, Y  +481.122, Z    +0.000, E1   +41.279, E3 +429008.899}
SPL {X  -162.820, Y  +478.698, Z    +0.000, E1   +40.526, E3 +429019.248}
SPL {X  -162.820, Y  +475.203, Z    +0.000, E1   +39.596, E3 +429033.708}
SPL {X  -162.820, Y  +472.097, Z    +0.000, E1   +38.411, E3 +429048.674}
SPL {X  -162.820, Y  +469.633, Z    +0.000, E1   +37.658, E3 +429059.750}
ENDSPLINE

SPLINE
SPL {X  -162.820, Y  +489.849, Z    +0.000, E1   +25.651, E3 +429072.843}
ENDSPLINE

SPLINE
SPL {X  -162.820, Y  +485.392, Z    +0.000, E1   +25.667, E3 +429092.061}
SPL {X  -162.820, Y  +482.092, Z    +0.000, E1   +25.593, E3 +429106.749}
SPL {X  -162.820, Y  +479.578, Z    +0.000, E1   +25.634, E3 +429117.392}
SPL {X  -162.820, Y  +476.226, Z    +0.000, E1   +25.672, E3 +429131.783}
SPL {X  -162.820, Y  +473.037, Z    +0.000, E1   +25.618, E3 +429145.873}
SPL {X  -162.820, Y  +470.744, Z    +0.000, E1   +25.641, E3 +429155.614}
SPL {X  -162.820, Y  +467.745, Z    +0.000, E1   +25.668, E3 +429168.596}
SPL {X  -162.820, Y  +463.978, Z    +0.000, E1   +25.651, E3 +429185.074}
SPL {X  -162.820, Y  +459.882, Z    +0.000, E1   +25.674, E3 +429202.708}
SPL {X  -162.820, Y  +456.773, Z    +0.000, E1   +25.591, E3 +429216.654}
SPL {X  -162.820, Y  +454.429, Z    +0.000, E1   +25.642, E3 +429226.422}
SPL {X  -162.820, Y  +451.204, Z    +0.000, E1   +25.672, E3 +429240.449}
SPL {X  -162.820, Y  +447.822, Z    +0.000, E1   +25.664, E3 +429254.933}
SPL {X  -162.820, Y  +445.556, Z    +0.000, E1   +25.626, E3 +429265.063}
SPL {X  -162.820, Y  +443.328, Z    +0.000, E1   +25.642, E3 +429274.578}
SPL {X  -162.820, Y  +440.857, Z    +0.000, E1   +25.614, E3 +429285.612}
SPL {X  -162.820, Y  +437.636, Z    +0.000, E1   +25.597, E3 +429299.776}
SPL {X  -162.820, Y  +434.768, Z    +0.000, E1   +25.655, E3 +429311.677}
SPL {X  -162.820, Y  +431.823, Z    +0.000, E1   +25.651, E3 +429324.676}
SPL {X  -162.820, Y  +427.740, Z    +0.000, E1   +25.667, E3 +429342.304}
SPL {X  -162.820, Y  +423.655, Z    +0.000, E1   +25.628, E3 +429360.328}
SPL {X  -162.820, Y  +419.407, Z    +0.000, E1   +25.665, E3 +429378.521}
SPL {X  -162.820, Y  +415.900, Z    +0.000, E1   +25.638, E3 +429393.790}
SPL {X  -162.820, Y  +413.088, Z    +0.000, E1   +25.644, E3 +429405.946}
SPL {X  -162.820, Y  +410.320, Z    +0.000, E1   +25.604, E3 +429418.265}
SPL {X  -162.820, Y  +407.487, Z    +0.000, E1   +25.617, E3 +429430.473}
SPL {X  -162.820, Y  +405.108, Z    +0.000, E1   +25.535, E3 +429441.441}
SPL {X  -162.820, Y  +401.373, Z    +0.000, E1   +25.736, E3 +429456.277}
SPL {X  -162.820, Y  +397.357, Z    +0.000, E1   +25.652, E3 +429474.347}
SPL {X  -162.820, Y  +393.659, Z    +0.000, E1   +25.666, E3 +429490.148}
SPL {X  -162.820, Y  +390.679, Z    +0.000, E1   +25.624, E3 +429503.391}
SPL {X  -162.820, Y  +387.939, Z    +0.000, E1   +25.627, E3 +429515.250}
SPL {X  -162.820, Y  +384.398, Z    +0.000, E1   +25.707, E3 +429530.148}
SPL {X  -162.820, Y  +380.448, Z    +0.000, E1   +25.674, E3 +429547.512}
SPL {X  -162.785, Y  +377.106, Z    +0.000, E1   +25.598, E3 +429562.456}
SPL {X  -162.709, Y  +374.484, Z    +0.000, E1   +25.711, E3 +429572.907}
SPL {X  -162.623, Y  +372.485, Z    +0.000, E1   +25.631, E3 +429582.187}
SPL {X  -162.487, Y  +370.088, Z    +0.000, E1   +25.525, E3 +429593.442}
SPL {X  -162.243, Y  +366.801, Z    +0.000, E1   +25.618, E3 +429607.082}
SPL {X  -161.977, Y  +363.953, Z    +0.000, E1   +25.528, E3 +429620.008}
SPL {X  -161.695, Y  +361.389, Z    +0.000, E1   +25.445, E3 +429631.824}
SPL {X  -161.364, Y  +358.774, Z    +0.000, E1   +25.454, E3 +429643.024}
SPL {X  -160.939, Y  +355.820, Z    +0.000, E1   +26.179, E3 +429650.242}
SPL {X  -155.035, Y  +330.756, Z    +0.000, E1   +37.918, E3 +429656.576}
SPL {X  -153.918, Y  +327.401, Z    +0.000, E1   +34.677, E3 +429691.877}
ENDSPLINE

SPLINE
SPL {X  -159.701, Y  +348.785, Z    +0.000, E1   +24.361, E3 +429699.358}
SPL {X  -162.442, Y  +369.407, Z    +0.000, E1   +11.234, E3 +429728.993}
SPL {X  -162.820, Y  +384.333, Z    +0.000, E1    +1.902, E3 +429730.199}
SPL {X  -162.820, Y  +389.940, Z    +0.000, E1    -2.281, E3 +429733.120}
SPL {X  -162.820, Y  +396.652, Z    +0.000, E1    -7.520, E3 +429732.699}
SPL {X  -162.820, Y  +406.605, Z    +0.000, E1   -16.760, E3 +429725.176}
SPL {X  -162.820, Y  +418.675, Z    +0.000, E1   -22.201, E3 +429751.424}
SPL {X  -162.820, Y  +425.113, Z    +0.000, E1   -25.243, E3 +429760.360}
SPL {X  -162.820, Y  +441.937, Z    +0.000, E1   -31.578, E3 +429782.439}
ENDSPLINE

SPLINE
SPL {X  -162.820, Y  +437.771, Z    +0.000, E1   -26.555, E3 +429801.539}
ENDSPLINE

SPLINE
SPL {X  -162.820, Y  +439.120, Z    +0.000, E1   -25.352, E3 +429816.082}
SPL {X  -162.820, Y  +441.593, Z    +0.000, E1   -25.391, E3 +429826.634}
SPL {X  -162.820, Y  +444.317, Z    +0.000, E1   -25.492, E3 +429837.815}
SPL {X  -162.820, Y  +446.544, Z    +0.000, E1   -25.427, E3 +429847.985}
SPL {X  -162.820, Y  +448.500, Z    +0.000, E1   -25.425, E3 +429856.586}
SPL {X  -162.820, Y  +451.056, Z    +0.000, E1   -25.443, E3 +429867.694}
SPL {X  -162.820, Y  +454.662, Z    +0.000, E1   -25.474, E3 +429883.438}
SPL {X  -162.820, Y  +458.079, Z    +0.000, E1   -25.369, E3 +429899.017}
SPL {X  -162.820, Y  +460.719, Z    +0.000, E1   -25.411, E3 +429910.275}
SPL {X  -162.820, Y  +463.419, Z    +0.000, E1   -25.510, E3 +429921.313}
SPL {X  -162.820, Y  +465.376, Z    +0.000, E1   -25.372, E3 +429930.901}
SPL {X  -162.820, Y  +467.440, Z    +0.000, E1   -25.427, E3 +429939.532}
SPL {X  -162.820, Y  +470.010, Z    +0.000, E1   -25.445, E3 +429950.737}
SPL {X  -162.820, Y  +473.445, Z    +0.000, E1   -25.493, E3 +429965.461}
SPL {X  -162.820, Y  +476.157, Z    +0.000, E1   -25.426, E3 +429977.676}
SPL {X  -162.820, Y  +478.461, Z    +0.000, E1   -25.410, E3 +429987.955}
SPL {X  -162.820, Y  +481.644, Z    +0.000, E1   -25.433, E3 +430001.902}
SPL {X  -162.820, Y  +486.042, Z    +0.000, E1   -25.483, E3 +430020.821}
SPL {X  -162.820, Y  +490.287, Z    +0.000, E1   -25.463, E3 +430039.540}
SPL {X  -162.820, Y  +494.454, Z    +0.000, E1   -25.465, E3 +430057.771}
SPL {X  -162.820, Y  +498.644, Z    +0.000, E1   -25.463, E3 +430076.147}
SPL {X  -162.820, Y  +502.845, Z    +0.000, E1   -25.458, E3 +430094.580}
SPL {X  -162.820, Y  +506.050, Z    +0.000, E1   -25.420, E3 +430108.720}
SPL {X  -162.820, Y  +508.346, Z    +0.000, E1   -25.444, E3 +430118.568}
SPL {X  -162.820, Y  +510.377, Z    +0.000, E1   -25.398, E3 +430127.814}
SPL {X  -162.820, Y  +513.176, Z    +0.000, E1   -25.443, E3 +430139.859}
SPL {X  -162.820, Y  +516.690, Z    +0.000, E1   -25.465, E3 +430155.070}
SPL {X  -162.820, Y  +519.134, Z    +0.000, E1   -25.366, E3 +430166.391}
SPL {X  -162.820, Y  +521.486, Z    +0.000, E1   -25.382, E3 +430176.687}
SPL {X  -162.820, Y  +524.180, Z    +0.000, E1   -25.495, E3 +430187.560}
SPL {X  -162.820, Y  +527.020, Z    +0.000, E1   -25.477, E3 +430200.253}
SPL {X  -162.820, Y  +529.670, Z    +0.000, E1   -25.472, E3 +430211.710}
SPL {X  -162.820, Y  +532.006, Z    +0.000, E1   -25.455, E3 +430222.167}
SPL {X  -162.820, Y  +534.806, Z    +0.000, E1   -25.465, E3 +430234.283}
SPL {X  -162.820, Y  +537.226, Z    +0.000, E1   -25.378, E3 +430245.565}
SPL {X  -162.820, Y  +540.345, Z    +0.000, E1   -25.451, E3 +430258.746}
SPL {X  -162.820, Y  +543.279, Z    +0.000, E1   -25.419, E3 +430271.779}
SPL {X  -162.820, Y  +546.125, Z    +0.000, E1   -25.505, E3 +430283.574}
SPL {X  -162.820, Y  +549.578, Z    +0.000, E1   -25.462, E3 +430299.198}
SPL {X  -162.820, Y  +553.157, Z    +0.000, E1   -25.443, E3 +430314.861}
SPL {X  -162.820, Y  +556.150, Z    +0.000, E1   -25.445, E3 +430327.951}
SPL {X  -162.820, Y  +559.215, Z    +0.000, E1   -25.460, E3 +430341.252}
SPL {X  -162.820, Y  +562.125, Z    +0.000, E1   -25.434, E3 +430354.173}
SPL {X  -162.820, Y  +564.880, Z    +0.000, E1   -25.448, E3 +430366.127}
SPL {X  -162.820, Y  +568.326, Z    +0.000, E1   -25.470, E3 +430381.186}
SPL {X  -162.820, Y  +571.303, Z    +0.000, E1   -25.427, E3 +430394.359}
SPL {X  -162.820, Y  +574.067, Z    +0.000, E1   -25.459, E3 +430406.298}
SPL {X  -162.820, Y  +576.597, Z    +0.000, E1   -25.400, E3 +430417.770}
SPL {X  -162.820, Y  +578.977, Z    +0.000, E1   -25.460, E3 +430427.702}
SPL {X  -162.820, Y  +581.995, Z    +0.000, E1   -25.468, E3 +430441.060}
SPL {X  -162.820, Y  +585.512, Z    +0.000, E1   -25.448, E3 +430456.484}
SPL {X  -162.820, Y  +588.371, Z    +0.000, E1   -25.460, E3 +430468.870}
SPL {X  -162.820, Y  +591.246, Z    +0.000, E1   -25.415, E3 +430481.889}
SPL {X  -162.820, Y  +594.339, Z    +0.000, E1   -25.487, E3 +430494.791}
SPL {X  -162.820, Y  +596.868, Z    +0.000, E1   -25.461, E3 +430506.054}
SPL {X  -162.820, Y  +599.135, Z    +0.000, E1   -25.398, E3 +430516.423}
SPL {X  -162.820, Y  +601.296, Z    +0.000, E1   -25.399, E3 +430525.905}
SPL {X  -162.820, Y  +603.808, Z    +0.000, E1   -25.554, E3 +430535.693}
SPL {X  -162.820, Y  +607.007, Z    +0.000, E1   -25.491, E3 +430550.384}
SPL {X  -162.820, Y  +611.438, Z    +0.000, E1   -25.467, E3 +430569.974}
SPL {X  -162.820, Y  +615.388, Z    +0.000, E1   -25.455, E3 +430587.233}
SPL {X  -162.820, Y  +618.103, Z    +0.000, E1   -25.456, E3 +430598.980}
SPL {X  -162.820, Y  +621.264, Z    +0.000, E1   -25.514, E3 +430612.583}
SPL {X  -162.820, Y  +624.430, Z    +0.000, E1   -25.475, E3 +430626.514}
SPL {X  -162.820, Y  +626.570, Z    +0.000, E1   -25.441, E3 +430636.114}
SPL {X  -162.820, Y  +628.902, Z    +0.000, E1   -25.449, E3 +430646.294}
SPL {X  -162.820, Y  +631.177, Z    +0.000, E1   -25.467, E3 +430656.126}
SPL {X  -162.820, Y  +633.994, Z    +0.000, E1   -25.503, E3 +430668.172}
SPL {X  -162.820, Y  +636.469, Z    +0.000, E1   -25.465, E3 +430679.216}
SPL {X  -162.820, Y  +638.486, Z    +0.000, E1   -25.456, E3 +430688.133}
SPL {X  -162.820, Y  +640.803, Z    +0.000, E1   -25.462, E3 +430698.195}
SPL {X  -162.820, Y  +643.028, Z    +0.000, E1   -25.494, E3 +430707.704}
SPL {X  -162.820, Y  +645.694, Z    +0.000, E1   -25.540, E3 +430718.992}
SPL {X  -162.820, Y  +649.102, Z    +0.000, E1   -25.495, E3 +430734.420}
SPL {X  -162.820, Y  +652.810, Z    +0.000, E1   -25.497, E3 +430750.453}
SPL {X  -162.820, Y  +655.214, Z    +0.000, E1   -25.485, E3 +430760.956}
SPL {X  -162.820, Y  +657.616, Z    +0.000, E1   -25.511, E3 +430771.310}
SPL {X  -162.820, Y  +660.007, Z    +0.000, E1   -25.550, E3 +430781.372}
SPL {X  -162.820, Y  +662.980, Z    +0.000, E1   -25.505, E3 +430794.930}
SPL {X  -162.820, Y  +667.253, Z    +0.000, E1   -25.483, E3 +430813.807}
SPL {X  -162.820, Y  +671.102, Z    +0.000, E1   -25.514, E3 +430830.257}
SPL {X  -162.820, Y  +673.648, Z    +0.000, E1   -25.431, E3 +430841.924}
SPL {X  -162.796, Y  +676.319, Z    +0.000, E1   -25.526, E3 +430852.934}
SPL {X  -162.739, Y  +678.625, Z    +0.000, E1   -25.423, E3 +430863.725}
SPL {X  -162.669, Y  +680.515, Z    +0.000, E1   -25.398, E3 +430872.179}
SPL {X  -162.545, Y  +682.952, Z    +0.000, E1   -25.510, E3 +430882.041}
SPL {X  -162.381, Y  +685.455, Z    +0.000, E1   -25.410, E3 +430893.728}
SPL {X  -162.194, Y  +687.760, Z    +0.000, E1   -25.360, E3 +430904.164}
SPL {X  -161.987, Y  +689.945, Z    +0.000, E1   -25.406, E3 +430913.316}
SPL {X  -161.711, Y  +692.468, Z    +0.000, E1   -25.300, E3 +430925.315}
SPL {X  -161.141, Y  +696.825, Z    +0.000, E1   -26.170, E3 +430937.449}
SPL {X  -157.976, Y  +712.921, Z    +0.000, E1   -33.197, E3 +430947.990}
ENDSPLINE

SPLINE
SPL {X  -160.738, Y  +699.453, Z    +0.000, E1   -21.994, E3 +430985.617}
SPL {X  -160.945, Y  +698.140, Z    +0.000, E1   -18.412, E3 +431027.856}
SPL {X  -162.497, Y  +683.755, Z    +0.000, E1   -10.754, E3 +431022.000}
SPL {X  -162.819, Y  +673.996, Z    +0.000, E1    -4.745, E3 +431021.601}
ENDSPLINE

SPLINE
SPL {X  -162.791, Y  +676.574, Z    +0.000, E1    -6.127, E3 +431034.289}
ENDSPLINE

SPLINE
SPL {X  -162.820, Y  +667.935, Z    +0.000, E1    -0.509, E3 +431024.375}
SPL {X  -162.820, Y  +662.949, Z    +0.000, E1    +3.113, E3 +431022.494}
SPL {X  -162.820, Y  +658.484, Z    +0.000, E1    +6.336, E3 +431029.639}
SPL {X  -162.820, Y  +640.102, Z    +0.000, E1   +22.409, E3 +431024.378}
SPL {X  -162.820, Y  +633.503, Z    +0.000, E1   +21.975, E3 +431056.614}
SPL {X  -162.820, Y  +611.299, Z    +0.000, E1   +31.088, E3 +431084.727}
ENDSPLINE

SPLINE
SPL {X  -162.820, Y  +618.877, Z    +0.000, E1   +25.259, E3 +431096.221}
ENDSPLINE

SPLINE
SPL {X  -162.820, Y  +617.582, Z    +0.000, E1   +24.552, E3 +431107.598}
SPL {X  -162.820, Y  +614.716, Z    +0.000, E1   +24.535, E3 +431120.810}
SPL {X  -162.820, Y  +611.754, Z    +0.000, E1   +24.563, E3 +431134.098}
SPL {X  -162.820, Y  +608.970, Z    +0.000, E1   +24.542, E3 +431146.938}
SPL {X  -162.820, Y  +606.285, Z    +0.000, E1   +24.533, E3 +431159.273}
SPL {X  -162.820, Y  +603.509, Z    +0.000, E1   +24.546, E3 +431171.811}
SPL {X  -162.820, Y  +600.818, Z    +0.000, E1   +24.590, E3 +431183.733}
SPL {X  -162.820, Y  +598.053, Z    +0.000, E1   +24.547, E3 +431196.716}
SPL {X  -162.820, Y  +595.188, Z    +0.000, E1   +24.538, E3 +431209.805}
SPL {X  -162.820, Y  +592.738, Z    +0.000, E1   +24.551, E3 +431220.853}
SPL {X  -162.820, Y  +590.118, Z    +0.000, E1   +24.544, E3 +431232.912}
SPL {X  -162.820, Y  +587.204, Z    +0.000, E1   +24.592, E3 +431245.789}
SPL {X  -162.820, Y  +584.766, Z    +0.000, E1   +24.499, E3 +431257.622}
SPL {X  -162.820, Y  +581.896, Z    +0.000, E1   +24.528, E3 +431270.564}
SPL {X  -162.820, Y  +579.244, Z    +0.000, E1   +24.610, E3 +431281.909}
SPL {X  -162.820, Y  +576.848, Z    +0.000, E1   +24.543, E3 +431293.450}
SPL {X  -162.820, Y  +573.694, Z    +0.000, E1   +24.535, E3 +431307.919}
SPL {X  -162.820, Y  +570.310, Z    +0.000, E1   +24.556, E3 +431323.236}
SPL {X  -162.820, Y  +567.494, Z    +0.000, E1   +24.547, E3 +431336.021}
SPL {X  -162.820, Y  +564.977, Z    +0.000, E1   +24.571, E3 +431347.351}
SPL {X  -162.820, Y  +562.356, Z    +0.000, E1   +24.575, E3 +431359.250}
SPL {X  -162.820, Y  +558.990, Z    +0.000, E1   +24.558, E3 +431374.900}
SPL {X  -162.820, Y  +555.584, Z    +0.000, E1   +24.559, E3 +431390.269}
SPL {X  -162.820, Y  +552.867, Z    +0.000, E1   +24.583, E3 +431402.464}
SPL {X  -162.820, Y  +549.589, Z    +0.000, E1   +24.547, E3 +431417.830}
SPL {X  -162.820, Y  +545.742, Z    +0.000, E1   +24.577, E3 +431435.117}
SPL {X  -162.820, Y  +542.142, Z    +0.000, E1   +24.582, E3 +431451.470}
SPL {X  -162.820, Y  +538.903, Z    +0.000, E1   +24.519, E3 +431466.686}
SPL {X  -162.820, Y  +536.451, Z    +0.000, E1   +24.519, E3 +431477.766}
SPL {X  -162.820, Y  +534.025, Z    +0.000, E1   +24.589, E3 +431488.366}
SPL {X  -162.820, Y  +531.527, Z    +0.000, E1   +24.582, E3 +431499.752}
SPL {X  -162.820, Y  +529.165, Z    +0.000, E1   +24.521, E3 +431511.000}
SPL {X  -162.820, Y  +525.802, Z    +0.000, E1   +24.585, E3 +431526.020}
SPL {X  -162.820, Y  +521.731, Z    +0.000, E1   +24.542, E3 +431544.957}
SPL {X  -162.820, Y  +518.185, Z    +0.000, E1   +24.561, E3 +431560.829}
SPL {X  -162.820, Y  +508.728, Z    +0.000, E1   +28.484, E3 +431571.368}
SPL {X  -162.820, Y  +500.664, Z    +0.000, E1   +31.476, E3 +431580.032}
SPL {X  -162.820, Y  +499.290, Z    +0.000, E1   +30.657, E3 +431590.315}
SPL {X  -162.820, Y  +497.251, Z    +0.000, E1   +29.634, E3 +431604.790}
SPL {X  -162.820, Y  +495.647, Z    +0.000, E1   +28.606, E3 +431617.666}
SPL {X  -162.820, Y  +494.678, Z    +0.000, E1   +27.647, E3 +431628.367}
SPL {X  -162.820, Y  +493.757, Z    +0.000, E1   +26.462, E3 +431640.727}
SPL {X  -162.820, Y  +491.420, Z    +0.000, E1   +25.780, E3 +431655.989}
SPL {X  -162.820, Y  +487.351, Z    +0.000, E1   +25.663, E3 +431674.505}
SPL {X  -162.820, Y  +484.247, Z    +0.000, E1   +25.651, E3 +431687.832}
SPL {X  -162.820, Y  +482.092, Z    +0.000, E1   +25.593, E3 +431697.659}
SPL {X  -162.820, Y  +479.578, Z    +0.000, E1   +25.634, E3 +431708.301}
SPL {X  -162.820, Y  +477.137, Z    +0.000, E1   +25.632, E3 +431718.881}
SPL {X  -162.820, Y  +473.770, Z    +0.000, E1   +25.664, E3 +431733.426}
SPL {X  -162.820, Y  +469.694, Z    +0.000, E1   +25.657, E3 +431751.157}
SPL {X  -162.820, Y  +465.727, Z    +0.000, E1   +25.676, E3 +431768.200}
SPL {X  -162.820, Y  +463.001, Z    +0.000, E1   +25.614, E3 +431780.317}
SPL {X  -162.820, Y  +459.882, Z    +0.000, E1   +25.674, E3 +431793.617}
SPL {X  -162.820, Y  +456.773, Z    +0.000, E1   +25.591, E3 +431807.563}
SPL {X  -162.820, Y  +454.429, Z    +0.000, E1   +25.642, E3 +431817.331}
SPL {X  -162.820, Y  +451.204, Z    +0.000, E1   +25.672, E3 +431831.358}
SPL {X  -162.820, Y  +447.822, Z    +0.000, E1   +25.664, E3 +431845.842}
SPL {X  -162.820, Y  +445.556, Z    +0.000, E1   +25.626, E3 +431855.972}
SPL {X  -162.820, Y  +442.508, Z    +0.000, E1   +25.657, E3 +431869.066}
SPL {X  -162.820, Y  +439.273, Z    +0.000, E1   +25.576, E3 +431883.704}
SPL {X  -162.820, Y  +436.773, Z    +0.000, E1   +25.602, E3 +431894.269}
SPL {X  -162.820, Y  +433.761, Z    +0.000, E1   +25.681, E3 +431906.947}
SPL {X  -162.820, Y  +430.942, Z    +0.000, E1   +25.597, E3 +431919.633}
SPL {X  -162.820, Y  +428.576, Z    +0.000, E1   +25.647, E3 +431929.570}
SPL {X  -162.820, Y  +426.525, Z    +0.000, E1   +25.610, E3 +431938.678}
SPL {X  -162.820, Y  +423.655, Z    +0.000, E1   +25.628, E3 +431951.237}
SPL {X  -162.820, Y  +419.407, Z    +0.000, E1   +25.665, E3 +431969.430}
SPL {X  -162.820, Y  +415.900, Z    +0.000, E1   +25.638, E3 +431984.699}
SPL {X  -162.820, Y  +413.088, Z    +0.000, E1   +25.644, E3 +431996.855}
SPL {X  -162.820, Y  +410.320, Z    +0.000, E1   +25.604, E3 +432009.174}
SPL {X  -162.820, Y  +407.487, Z    +0.000, E1   +25.617, E3 +432021.382}
SPL {X  -162.820, Y  +405.108, Z    +0.000, E1   +25.535, E3 +432032.350}
SPL {X  -162.820, Y  +401.373, Z    +0.000, E1   +25.736, E3 +432047.186}
SPL {X  -162.820, Y  +397.357, Z    +0.000, E1   +25.652, E3 +432065.256}
SPL {X  -162.820, Y  +393.659, Z    +0.000, E1   +25.666, E3 +432081.057}
SPL {X  -162.820, Y  +390.679, Z    +0.000, E1   +25.624, E3 +432094.300}
SPL {X  -162.820, Y  +387.939, Z    +0.000, E1   +25.627, E3 +432106.159}
SPL {X  -162.820, Y  +384.398, Z    +0.000, E1   +25.707, E3 +432121.057}
SPL {X  -162.820, Y  +380.448, Z    +0.000, E1   +25.674, E3 +432138.421}
SPL {X  -162.785, Y  +377.106, Z    +0.000, E1   +25.598, E3 +432153.365}
SPL {X  -162.709, Y  +374.484, Z    +0.000, E1   +25.711, E3 +432163.816}
SPL {X  -162.623, Y  +372.485, Z    +0.000, E1   +25.631, E3 +432173.097}
SPL {X  -162.487, Y  +370.088, Z    +0.000, E1   +25.525, E3 +432184.351}
SPL {X  -162.243, Y  +366.801, Z    +0.000, E1   +25.618, E3 +432197.991}
SPL {X  -161.977, Y  +363.953, Z    +0.000, E1   +25.528, E3 +432210.917}
SPL {X  -161.695, Y  +361.389, Z    +0.000, E1   +25.445, E3 +432222.733}
SPL {X  -161.190, Y  +357.520, Z    +0.000, E1   +25.774, E3 +432236.984}
SPL {X  -155.035, Y  +330.756, Z    +0.000, E1   +37.918, E3 +432247.485}
SPL {X  -153.918, Y  +327.401, Z    +0.000, E1   +34.677, E3 +432282.786}
ENDSPLINE

SPLINE
SPL {X  -159.701, Y  +348.785, Z    +0.000, E1   +24.361, E3 +432290.267}
SPL {X  -161.904, Y  +363.251, Z    +0.000, E1   +14.606, E3 +432320.062}
SPL {X  -162.745, Y  +375.561, Z    +0.000, E1    +7.538, E3 +432320.258}
SPL {X  -162.820, Y  +385.424, Z    +0.000, E1    +1.080, E3 +432321.153}
SPL {X  -162.820, Y  +389.940, Z    +0.000, E1    -2.281, E3 +432324.029}
SPL {X  -162.820, Y  +396.652, Z    +0.000, E1    -7.520, E3 +432323.608}
SPL {X  -162.820, Y  +406.605, Z    +0.000, E1   -16.760, E3 +432316.085}
SPL {X  -162.820, Y  +418.675, Z    +0.000, E1   -22.201, E3 +432342.333}
SPL {X  -162.820, Y  +425.113, Z    +0.000, E1   -25.243, E3 +432351.269}
SPL {X  -162.820, Y  +441.937, Z    +0.000, E1   -31.578, E3 +432373.348}
ENDSPLINE

SPLINE
SPL {X  -162.820, Y  +437.771, Z    +0.000, E1   -26.555, E3 +432392.448}
ENDSPLINE

SPLINE
SPL {X  -162.820, Y  +439.120, Z    +0.000, E1   -25.352, E3 +432406.991}
SPL {X  -162.820, Y  +441.593, Z    +0.000, E1   -25.391, E3 +432417.543}
SPL {X  -162.820, Y  +444.317, Z    +0.000, E1   -25.492, E3 +432428.724}
SPL {X  -162.820, Y  +446.544, Z    +0.000, E1   -25.427, E3 +432438.894}
SPL {X  -162.820, Y  +448.500, Z    +0.000, E1   -25.425, E3 +432447.495}
SPL {X  -162.820, Y  +451.056, Z    +0.000, E1   -25.443, E3 +432458.603}
SPL {X  -162.820, Y  +454.662, Z    +0.000, E1   -25.474, E3 +432474.347}
SPL {X  -162.820, Y  +458.079, Z    +0.000, E1   -25.369, E3 +432489.926}
SPL {X  -162.820, Y  +460.719, Z    +0.000, E1   -25.411, E3 +432501.184}
SPL {X  -162.820, Y  +463.419, Z    +0.000, E1   -25.510, E3 +432512.222}
SPL {X  -162.820, Y  +466.458, Z    +0.000, E1   -25.433, E3 +432526.278}
SPL {X  -162.820, Y  +470.010, Z    +0.000, E1   -25.445, E3 +432541.646}
SPL {X  -162.820, Y  +472.345, Z    +0.000, E1   -25.448, E3 +432551.733}
SPL {X  -162.820, Y  +475.191, Z    +0.000, E1   -25.489, E3 +432564.095}
SPL {X  -162.820, Y  +478.461, Z    +0.000, E1   -25.410, E3 +432578.865}
SPL {X  -162.820, Y  +480.780, Z    +0.000, E1   -25.447, E3 +432588.726}
SPL {X  -162.820, Y  +483.622, Z    +0.000, E1   -25.381, E3 +432601.768}
SPL {X  -162.820, Y  +487.570, Z    +0.000, E1   -25.482, E3 +432618.406}
SPL {X  -162.820, Y  +491.017, Z    +0.000, E1   -25.445, E3 +432633.621}
SPL {X  -162.820, Y  +493.705, Z    +0.000, E1   -25.443, E3 +432645.405}
SPL {X  -162.820, Y  +497.247, Z    +0.000, E1   -25.470, E3 +432660.867}
SPL {X  -162.820, Y  +501.343, Z    +0.000, E1   -25.435, E3 +432679.066}
SPL {X  -162.820, Y  +505.370, Z    +0.000, E1   -25.456, E3 +432696.530}
SPL {X  -162.820, Y  +509.412, Z    +0.000, E1   -25.458, E3 +432714.253}
SPL {X  -162.820, Y  +512.406, Z    +0.000, E1   -25.425, E3 +432727.409}
SPL {X  -162.820, Y  +515.039, Z    +0.000, E1   -25.452, E3 +432738.819}
SPL {X  -162.820, Y  +518.350, Z    +0.000, E1   -25.425, E3 +432753.569}
SPL {X  -162.820, Y  +521.486, Z    +0.000, E1   -25.382, E3 +432767.597}
SPL {X  -162.820, Y  +524.180, Z    +0.000, E1   -25.495, E3 +432778.469}
SPL {X  -162.820, Y  +527.020, Z    +0.000, E1   -25.477, E3 +432791.162}
SPL {X  -162.820, Y  +529.670, Z    +0.000, E1   -25.472, E3 +432802.619}
SPL {X  -162.820, Y  +532.006, Z    +0.000, E1   -25.455, E3 +432813.076}
SPL {X  -162.820, Y  +534.806, Z    +0.000, E1   -25.465, E3 +432825.193}
SPL {X  -162.820, Y  +537.226, Z    +0.000, E1   -25.378, E3 +432836.474}
SPL {X  -162.820, Y  +540.345, Z    +0.000, E1   -25.451, E3 +432849.655}
SPL {X  -162.820, Y  +543.279, Z    +0.000, E1   -25.419, E3 +432862.688}
SPL {X  -162.820, Y  +546.125, Z    +0.000, E1   -25.505, E3 +432874.483}
SPL {X  -162.820, Y  +548.232, Z    +0.000, E1   -25.424, E3 +432884.245}
SPL {X  -162.820, Y  +550.399, Z    +0.000, E1   -25.424, E3 +432893.796}
SPL {X  -162.820, Y  +553.157, Z    +0.000, E1   -25.443, E3 +432905.770}
SPL {X  -162.820, Y  +556.150, Z    +0.000, E1   -25.445, E3 +432918.860}
SPL {X  -162.820, Y  +559.215, Z    +0.000, E1   -25.460, E3 +432932.162}
SPL {X  -162.820, Y  +562.125, Z    +0.000, E1   -25.434, E3 +432945.082}
SPL {X  -162.820, Y  +564.880, Z    +0.000, E1   -25.448, E3 +432957.036}
SPL {X  -162.820, Y  +568.326, Z    +0.000, E1   -25.470, E3 +432972.095}
SPL {X  -162.820, Y  +571.303, Z    +0.000, E1   -25.427, E3 +432985.268}
SPL {X  -162.820, Y  +574.067, Z    +0.000, E1   -25.459, E3 +432997.207}
SPL {X  -162.820, Y  +576.597, Z    +0.000, E1   -25.400, E3 +433008.679}
SPL {X  -162.820, Y  +580.038, Z    +0.000, E1   -25.473, E3 +433023.374}
SPL {X  -162.820, Y  +583.044, Z    +0.000, E1   -25.450, E3 +433036.497}
SPL {X  -162.820, Y  +585.512, Z    +0.000, E1   -25.448, E3 +433047.393}
SPL {X  -162.820, Y  +588.371, Z    +0.000, E1   -25.460, E3 +433059.779}
SPL {X  -162.820, Y  +591.246, Z    +0.000, E1   -25.415, E3 +433072.798}
SPL {X  -162.820, Y  +594.339, Z    +0.000, E1   -25.487, E3 +433085.700}
SPL {X  -162.820, Y  +596.868, Z    +0.000, E1   -25.461, E3 +433096.964}
SPL {X  -162.820, Y  +599.135, Z    +0.000, E1   -25.398, E3 +433107.333}
SPL {X  -162.820, Y  +601.296, Z    +0.000, E1   -25.399, E3 +433116.814}
SPL {X  -162.820, Y  +604.526, Z    +0.000, E1   -25.502, E3 +433130.308}
SPL {X  -162.820, Y  +607.811, Z    +0.000, E1   -25.507, E3 +433144.523}
SPL {X  -162.820, Y  +610.517, Z    +0.000, E1   -25.412, E3 +433157.085}
SPL {X  -162.820, Y  +613.762, Z    +0.000, E1   -25.472, E3 +433170.892}
SPL {X  -162.820, Y  +616.216, Z    +0.000, E1   -25.419, E3 +433181.887}
SPL {X  -162.820, Y  +618.995, Z    +0.000, E1   -25.483, E3 +433193.737}
SPL {X  -162.820, Y  +622.118, Z    +0.000, E1   -25.492, E3 +433207.202}
SPL {X  -162.820, Y  +624.430, Z    +0.000, E1   -25.475, E3 +433217.423}
SPL {X  -162.820, Y  +626.570, Z    +0.000, E1   -25.441, E3 +433227.023}
SPL {X  -162.820, Y  +628.902, Z    +0.000, E1   -25.449, E3 +433237.203}
SPL {X  -162.820, Y  +631.177, Z    +0.000, E1   -25.467, E3 +433247.035}
SPL {X  -162.820, Y  +633.994, Z    +0.000, E1   -25.503, E3 +433259.081}
SPL {X  -162.820, Y  +637.619, Z    +0.000, E1   -25.497, E3 +433275.141}
SPL {X  -162.820, Y  +640.803, Z    +0.000, E1   -25.462, E3 +433289.104}
SPL {X  -162.820, Y  +643.028, Z    +0.000, E1   -25.494, E3 +433298.613}
SPL {X  -162.820, Y  +645.694, Z    +0.000, E1   -25.540, E3 +433309.901}
SPL {X  -162.820, Y  +649.102, Z    +0.000, E1   -25.495, E3 +433325.329}
SPL {X  -162.820, Y  +652.810, Z    +0.000, E1   -25.497, E3 +433341.362}
SPL {X  -162.820, Y  +655.214, Z    +0.000, E1   -25.485, E3 +433351.865}
SPL {X  -162.820, Y  +657.616, Z    +0.000, E1   -25.511, E3 +433362.219}
SPL {X  -162.820, Y  +660.851, Z    +0.000, E1   -25.520, E3 +433376.362}
SPL {X  -162.820, Y  +663.853, Z    +0.000, E1   -25.496, E3 +433389.544}
SPL {X  -162.820, Y  +666.096, Z    +0.000, E1   -25.408, E3 +433400.011}
SPL {X  -162.820, Y  +669.195, Z    +0.000, E1   -25.525, E3 +433412.848}
SPL {X  -162.820, Y  +672.979, Z    +0.000, E1   -25.478, E3 +433429.698}
SPL {X  -162.796, Y  +676.319, Z    +0.000, E1   -25.526, E3 +433443.843}
SPL {X  -162.707, Y  +679.552, Z    +0.000, E1   -25.443, E3 +433458.717}
SPL {X  -162.545, Y  +682.952, Z    +0.000, E1   -25.510, E3 +433472.950}
SPL {X  -162.381, Y  +685.455, Z    +0.000, E1   -25.410, E3 +433484.637}
SPL {X  -162.102, Y  +688.774, Z    +0.000, E1   -25.417, E3 +433499.251}
SPL {X  -161.711, Y  +692.468, Z    +0.000, E1   -25.300, E3 +433516.224}
SPL {X  -160.732, Y  +699.494, Z    +0.000, E1   -27.462, E3 +433529.697}
SPL {X  -157.189, Y  +715.948, Z    +0.000, E1   -34.218, E3 +433541.854}
ENDSPLINE

SPLINE
SPL {X  -157.848, Y  +713.428, Z    +0.000, E1   -28.857, E3 +433575.994}
SPL {X  -161.246, Y  +696.087, Z    +0.000, E1   -20.259, E3 +433574.674}
ENDSPLINE

SPLINE
SPL {X  -160.474, Y  +701.038, Z    +0.000, E1   -20.238, E3 +433613.046}
ENDSPLINE

SPLINE
SPL {X  -162.192, Y  +687.790, Z    +0.000, E1   -12.981, E3 +433614.552}
SPL {X  -162.807, Y  +675.545, Z    +0.000, E1    -5.787, E3 +433612.095}
ENDSPLINE

SPLINE
SPL {X  -162.791, Y  +676.574, Z    +0.000, E1    -6.127, E3 +433625.198}
ENDSPLINE

SPLINE
SPL {X  -162.820, Y  +666.063, Z    +0.000, E1    +0.780, E3 +433613.292}
SPL {X  -162.820, Y  +659.251, Z    +0.000, E1    +5.716, E3 +433619.508}
SPL {X  -162.820, Y  +640.102, Z    +0.000, E1   +22.409, E3 +433615.287}
SPL {X  -162.820, Y  +633.503, Z    +0.000, E1   +21.975, E3 +433647.524}
SPL {X  -162.820, Y  +611.299, Z    +0.000, E1   +31.088, E3 +433675.636}
ENDSPLINE

SPLINE
SPL {X  -162.820, Y  +618.877, Z    +0.000, E1   +25.259, E3 +433687.130}
ENDSPLINE

SPLINE
SPL {X  -162.820, Y  +617.582, Z    +0.000, E1   +24.552, E3 +433698.507}
SPL {X  -162.820, Y  +614.716, Z    +0.000, E1   +24.535, E3 +433711.719}
SPL {X  -162.820, Y  +611.754, Z    +0.000, E1   +24.563, E3 +433725.007}
SPL {X  -162.820, Y  +608.970, Z    +0.000, E1   +24.542, E3 +433737.847}
SPL {X  -162.820, Y  +606.285, Z    +0.000, E1   +24.533, E3 +433750.182}
SPL {X  -162.820, Y  +603.509, Z    +0.000, E1   +24.546, E3 +433762.720}
SPL {X  -162.820, Y  +600.818, Z    +0.000, E1   +24.590, E3 +433774.643}
SPL {X  -162.820, Y  +598.053, Z    +0.000, E1   +24.547, E3 +433787.626}
SPL {X  -162.820, Y  +595.188, Z    +0.000, E1   +24.538, E3 +433800.714}
SPL {X  -162.820, Y  +592.738, Z    +0.000, E1   +24.551, E3 +433811.762}
SPL {X  -162.820, Y  +590.118, Z    +0.000, E1   +24.544, E3 +433823.821}
SPL {X  -162.820, Y  +587.204, Z    +0.000, E1   +24.592, E3 +433836.698}
SPL {X  -162.820, Y  +584.766, Z    +0.000, E1   +24.499, E3 +433848.531}
SPL {X  -162.820, Y  +581.896, Z    +0.000, E1   +24.528, E3 +433861.473}
SPL {X  -162.820, Y  +579.244, Z    +0.000, E1   +24.610, E3 +433872.818}
SPL {X  -162.820, Y  +576.848, Z    +0.000, E1   +24.543, E3 +433884.359}
SPL {X  -162.820, Y  +573.694, Z    +0.000, E1   +24.535, E3 +433898.829}
SPL {X  -162.820, Y  +570.310, Z    +0.000, E1   +24.556, E3 +433914.145}
SPL {X  -162.820, Y  +567.494, Z    +0.000, E1   +24.547, E3 +433926.930}
SPL {X  -162.820, Y  +564.977, Z    +0.000, E1   +24.571, E3 +433938.260}
SPL {X  -162.820, Y  +562.356, Z    +0.000, E1   +24.575, E3 +433950.159}
SPL {X  -162.820, Y  +558.990, Z    +0.000, E1   +24.558, E3 +433965.809}
SPL {X  -162.820, Y  +555.584, Z    +0.000, E1   +24.559, E3 +433981.178}
SPL {X  -162.820, Y  +552.867, Z    +0.000, E1   +24.583, E3 +433993.373}
SPL {X  -162.820, Y  +549.589, Z    +0.000, E1   +24.547, E3 +434008.739}
SPL {X  -162.820, Y  +545.742, Z    +0.000, E1   +24.577, E3 +434026.026}
SPL {X  -162.820, Y  +542.142, Z    +0.000, E1   +24.582, E3 +434042.379}
SPL {X  -162.820, Y  +538.903, Z    +0.000, E1   +24.519, E3 +434057.595}
SPL {X  -162.820, Y  +536.451, Z    +0.000, E1   +24.519, E3 +434068.675}
SPL {X  -162.820, Y  +534.025, Z    +0.000, E1   +24.589, E3 +434079.275}
SPL {X  -162.820, Y  +531.527, Z    +0.000, E1   +24.582, E3 +434090.661}
SPL {X  -162.820, Y  +529.165, Z    +0.000, E1   +24.521, E3 +434101.910}
SPL {X  -162.820, Y  +526.822, Z    +0.000, E1   +24.559, E3 +434112.273}
SPL {X  -162.820, Y  +524.112, Z    +0.000, E1   +24.542, E3 +434124.890}
SPL {X  -162.820, Y  +521.048, Z    +0.000, E1   +24.515, E3 +434139.027}
SPL {X  -162.820, Y  +518.185, Z    +0.000, E1   +24.561, E3 +434151.738}
SPL {X  -162.820, Y  +508.728, Z    +0.000, E1   +28.484, E3 +434162.278}
SPL {X  -162.820, Y  +500.664, Z    +0.000, E1   +31.476, E3 +434170.942}
SPL {X  -162.820, Y  +499.290, Z    +0.000, E1   +30.657, E3 +434181.224}
SPL {X  -162.820, Y  +497.251, Z    +0.000, E1   +29.634, E3 +434195.699}
SPL {X  -162.820, Y  +495.647, Z    +0.000, E1   +28.606, E3 +434208.576}
SPL {X  -162.820, Y  +494.678, Z    +0.000, E1   +27.647, E3 +434219.276}
SPL {X  -162.820, Y  +493.757, Z    +0.000, E1   +26.462, E3 +434231.636}
SPL {X  -162.820, Y  +491.420, Z    +0.000, E1   +25.780, E3 +434246.898}
SPL {X  -162.820, Y  +487.351, Z    +0.000, E1   +25.663, E3 +434265.414}
SPL {X  -162.820, Y  +484.247, Z    +0.000, E1   +25.651, E3 +434278.741}
SPL {X  -162.820, Y  +482.092, Z    +0.000, E1   +25.593, E3 +434288.568}
SPL {X  -162.820, Y  +479.578, Z    +0.000, E1   +25.634, E3 +434299.210}
SPL {X  -162.820, Y  +477.137, Z    +0.000, E1   +25.632, E3 +434309.790}
SPL {X  -162.820, Y  +473.770, Z    +0.000, E1   +25.664, E3 +434324.335}
SPL {X  -162.820, Y  +469.694, Z    +0.000, E1   +25.657, E3 +434342.067}
SPL {X  -162.820, Y  +465.727, Z    +0.000, E1   +25.676, E3 +434359.110}
SPL {X  -162.820, Y  +461.675, Z    +0.000, E1   +25.655, E3 +434376.916}
SPL {X  -162.820, Y  +457.479, Z    +0.000, E1   +25.656, E3 +434395.096}
SPL {X  -162.820, Y  +453.678, Z    +0.000, E1   +25.652, E3 +434411.548}
SPL {X  -162.820, Y  +450.466, Z    +0.000, E1   +25.644, E3 +434425.493}
SPL {X  -162.820, Y  +447.822, Z    +0.000, E1   +25.664, E3 +434436.751}
SPL {X  -162.820, Y  +445.556, Z    +0.000, E1   +25.626, E3 +434446.882}
SPL {X  -162.820, Y  +442.508, Z    +0.000, E1   +25.657, E3 +434459.975}
SPL {X  -162.820, Y  +439.273, Z    +0.000, E1   +25.576, E3 +434474.613}
SPL {X  -162.820, Y  +436.773, Z    +0.000, E1   +25.602, E3 +434485.178}
SPL {X  -162.820, Y  +433.761, Z    +0.000, E1   +25.681, E3 +434497.857}
SPL {X  -162.820, Y  +430.942, Z    +0.000, E1   +25.597, E3 +434510.542}
SPL {X  -162.820, Y  +428.576, Z    +0.000, E1   +25.647, E3 +434520.480}
SPL {X  -162.820, Y  +425.120, Z    +0.000, E1   +25.647, E3 +434535.664}
SPL {X  -162.820, Y  +420.840, Z    +0.000, E1   +25.658, E3 +434554.170}
SPL {X  -162.820, Y  +416.590, Z    +0.000, E1   +25.659, E3 +434572.614}
SPL {X  -162.820, Y  +412.302, Z    +0.000, E1   +25.662, E3 +434591.220}
SPL {X  -162.820, Y  +408.133, Z    +0.000, E1   +25.637, E3 +434609.478}
SPL {X  -162.820, Y  +404.293, Z    +0.000, E1   +25.628, E3 +434626.201}
SPL {X  -162.820, Y  +400.835, Z    +0.000, E1   +25.694, E3 +434640.600}
SPL {X  -162.820, Y  +398.703, Z    +0.000, E1   +25.586, E3 +434650.592}
SPL {X  -162.820, Y  +395.582, Z    +0.000, E1   +25.684, E3 +434663.584}
SPL {X  -162.820, Y  +391.417, Z    +0.000, E1   +25.659, E3 +434681.922}
SPL {X  -162.820, Y  +387.939, Z    +0.000, E1   +25.627, E3 +434697.069}
SPL {X  -162.820, Y  +385.565, Z    +0.000, E1   +25.686, E3 +434706.857}
SPL {X  -162.820, Y  +383.458, Z    +0.000, E1   +25.657, E3 +434716.221}
SPL {X  -162.820, Y  +381.229, Z    +0.000, E1   +25.660, E3 +434725.897}
SPL {X  -162.797, Y  +377.786, Z    +0.000, E1   +25.638, E3 +434741.186}
SPL {X  -162.663, Y  +373.346, Z    +0.000, E1   +25.707, E3 +434759.925}
SPL {X  -162.487, Y  +370.088, Z    +0.000, E1   +25.525, E3 +434775.260}
SPL {X  -162.307, Y  +367.587, Z    +0.000, E1   +25.577, E3 +434785.678}
SPL {X  -162.041, Y  +364.588, Z    +0.000, E1   +25.591, E3 +434798.756}
SPL {X  -161.695, Y  +361.389, Z    +0.000, E1   +25.445, E3 +434813.642}
SPL {X  -161.364, Y  +358.774, Z    +0.000, E1   +25.454, E3 +434824.842}
SPL {X  -160.939, Y  +355.820, Z    +0.000, E1   +26.179, E3 +434832.060}
SPL {X  -155.035, Y  +330.756, Z    +0.000, E1   +37.918, E3 +434838.394}
SPL {X  -153.918, Y  +327.401, Z    +0.000, E1   +34.677, E3 +434873.695}
ENDSPLINE

